   SPTP {A1 7.169, A2 -36.078, A3 70.084, A4 37.543, A5 -95.645, A6 0.000, E1 1384.1, E2 0, E3 0, E4 0, E5 0, E6 0} C_DIS
   SPTP {A1 7.435, A2 -36.403, A3 70.202, A4 38.822, A5 -95.236, A6 0.000, E1 1384.19, E2 0, E3 0, E4 0, E5 0, E6 0} C_DIS
   SPTP {A1 7.436, A2 -36.388, A3 70.184, A4 38.835, A5 -95.248, A6 0.000, E1 1384.17, E2 0, E3 0, E4 0, E5 0, E6 0} C_DIS
   SPTP {A1 7.884, A2 -36.920, A3 70.315, A4 41.034, A5 -94.543, A6 0.000, E1 1384.27, E2 0, E3 0, E4 0, E5 0, E6 0} C_DIS
   SPTP {A1 8.287, A2 -37.697, A3 70.867, A4 43.097, A5 -93.668, A6 0.000, E1 1384.12, E2 0, E3 0, E4 0, E5 0, E6 0} C_DIS
   SPTP {A1 8.650, A2 -38.713, A3 71.817, A4 45.038, A5 -92.609, A6 0.000, E1 1383.69, E2 0, E3 0, E4 0, E5 0, E6 0} C_DIS
   SPTP {A1 9.006, A2 -39.694, A3 72.658, A4 46.997, A5 -91.531, A6 0.000, E1 1383.19, E2 0, E3 0, E4 0, E5 0, E6 0} C_DIS
   SPTP {A1 9.354, A2 -40.644, A3 73.399, A4 48.977, A5 -90.438, A6 0.000, E1 1382.62, E2 0, E3 0, E4 0, E5 0, E6 0} C_DIS
   SPTP {A1 9.691, A2 -41.569, A3 74.056, A4 50.968, A5 -89.331, A6 0.000, E1 1382, E2 0, E3 0, E4 0, E5 0, E6 0} C_DIS
   SPTP {A1 10.017, A2 -42.476, A3 74.643, A4 52.966, A5 -88.208, A6 0.000, E1 1381.33, E2 0, E3 0, E4 0, E5 0, E6 0} C_DIS
   SPTP {A1 10.328, A2 -43.371, A3 75.171, A4 54.967, A5 -87.068, A6 0.000, E1 1380.62, E2 0, E3 0, E4 0, E5 0, E6 0} C_DIS
   SPTP {A1 10.624, A2 -44.257, A3 75.647, A4 56.970, A5 -85.911, A6 0.000, E1 1379.87, E2 0, E3 0, E4 0, E5 0, E6 0} C_DIS
   SPTP {A1 10.880, A2 -45.245, A3 76.287, A4 58.874, A5 -84.671, A6 0.000, E1 1378.9, E2 0, E3 0, E4 0, E5 0, E6 0} C_DIS
   SPTP {A1 11.110, A2 -46.270, A3 76.958, A4 60.747, A5 -83.381, A6 0.000, E1 1377.81, E2 0, E3 0, E4 0, E5 0, E6 0} C_DIS
   SPTP {A1 11.327, A2 -47.266, A3 77.541, A4 62.657, A5 -82.098, A6 0.000, E1 1376.63, E2 0, E3 0, E4 0, E5 0, E6 0} C_DIS
   SPTP {A1 11.525, A2 -48.255, A3 78.076, A4 64.580, A5 -80.798, A6 0.000, E1 1375.41, E2 0, E3 0, E4 0, E5 0, E6 0} C_DIS
   SPTP {A1 11.705, A2 -49.225, A3 78.545, A4 66.533, A5 -79.499, A6 0.000, E1 1374.11, E2 0, E3 0, E4 0, E5 0, E6 0} C_DIS
   SPTP {A1 11.864, A2 -50.188, A3 78.970, A4 68.504, A5 -78.190, A6 0.000, E1 1372.75, E2 0, E3 0, E4 0, E5 0, E6 0} C_DIS
   SPTP {A1 12.001, A2 -51.135, A3 79.340, A4 70.506, A5 -76.884, A6 0.000, E1 1371.32, E2 0, E3 0, E4 0, E5 0, E6 0} C_DIS
   SPTP {A1 12.116, A2 -52.065, A3 79.653, A4 72.544, A5 -75.587, A6 0.000, E1 1369.81, E2 0, E3 0, E4 0, E5 0, E6 0} C_DIS
   SPTP {A1 12.207, A2 -52.982, A3 79.919, A4 74.615, A5 -74.295, A6 0.000, E1 1368.22, E2 0, E3 0, E4 0, E5 0, E6 0} C_DIS
   SPTP {A1 12.274, A2 -53.871, A3 80.119, A4 76.738, A5 -73.033, A6 0.000, E1 1366.55, E2 0, E3 0, E4 0, E5 0, E6 0} C_DIS
   SPTP {A1 12.314, A2 -54.747, A3 80.275, A4 78.900, A5 -71.783, A6 0.000, E1 1364.79, E2 0, E3 0, E4 0, E5 0, E6 0} C_DIS
   SPTP {A1 12.330, A2 -55.585, A3 80.354, A4 81.129, A5 -70.586, A6 0.000, E1 1362.92, E2 0, E3 0, E4 0, E5 0, E6 0} C_DIS
   SPTP {A1 12.318, A2 -56.405, A3 80.388, A4 83.407, A5 -69.414, A6 0.000, E1 1360.97, E2 0, E3 0, E4 0, E5 0, E6 0} C_DIS
   SPTP {A1 12.280, A2 -57.171, A3 80.349, A4 85.710, A5 -68.323, A6 0.000, E1 1358.99, E2 0, E3 0, E4 0, E5 0, E6 0} C_DIS
   SPTP {A1 12.211, A2 -57.855, A3 80.301, A4 87.795, A5 -67.313, A6 0.000, E1 1357.48, E2 0, E3 0, E4 0, E5 0, E6 0} C_DIS
   SPTP {A1 12.118, A2 -58.515, A3 80.224, A4 89.903, A5 -66.338, A6 0.000, E1 1355.95, E2 0, E3 0, E4 0, E5 0, E6 0} C_DIS
   SPTP {A1 12.001, A2 -59.157, A3 80.116, A4 92.058, A5 -65.395, A6 0.000, E1 1354.35, E2 0, E3 0, E4 0, E5 0, E6 0} C_DIS
   SPTP {A1 11.859, A2 -59.776, A3 79.972, A4 94.265, A5 -64.496, A6 0.000, E1 1352.66, E2 0, E3 0, E4 0, E5 0, E6 0} C_DIS
   SPTP {A1 11.695, A2 -60.368, A3 79.786, A4 96.528, A5 -63.651, A6 0.000, E1 1350.9, E2 0, E3 0, E4 0, E5 0, E6 0} C_DIS
   SPTP {A1 11.508, A2 -60.930, A3 79.557, A4 98.848, A5 -62.868, A6 0.000, E1 1349.05, E2 0, E3 0, E4 0, E5 0, E6 0} C_DIS
   SPTP {A1 11.299, A2 -61.454, A3 79.275, A4 101.229, A5 -62.166, A6 0.000, E1 1347.13, E2 0, E3 0, E4 0, E5 0, E6 0} C_DIS
   SPTP {A1 11.071, A2 -61.939, A3 78.958, A4 103.616, A5 -61.537, A6 0.000, E1 1345.24, E2 0, E3 0, E4 0, E5 0, E6 0} C_DIS
   SPTP {A1 10.826, A2 -62.433, A3 78.899, A4 105.464, A5 -60.737, A6 0.000, E1 1344.4, E2 0, E3 0, E4 0, E5 0, E6 0} C_DIS
   SPTP {A1 10.563, A2 -62.914, A3 78.831, A4 107.350, A5 -59.960, A6 0.000, E1 1343.51, E2 0, E3 0, E4 0, E5 0, E6 0} C_DIS
   SPTP {A1 10.285, A2 -63.380, A3 78.749, A4 109.279, A5 -59.216, A6 0.000, E1 1342.58, E2 0, E3 0, E4 0, E5 0, E6 0} C_DIS
   SPTP {A1 9.993, A2 -63.822, A3 78.643, A4 111.251, A5 -58.522, A6 0.000, E1 1341.59, E2 0, E3 0, E4 0, E5 0, E6 0} C_DIS
   SPTP {A1 9.691, A2 -64.237, A3 78.507, A4 113.267, A5 -57.891, A6 0.000, E1 1340.57, E2 0, E3 0, E4 0, E5 0, E6 0} C_DIS
   SPTP {A1 9.380, A2 -64.621, A3 78.337, A4 115.323, A5 -57.335, A6 0.000, E1 1339.52, E2 0, E3 0, E4 0, E5 0, E6 0} C_DIS
   SPTP {A1 9.064, A2 -65.063, A3 78.450, A4 116.938, A5 -56.526, A6 0.000, E1 1339.23, E2 0, E3 0, E4 0, E5 0, E6 0} C_DIS
   SPTP {A1 8.744, A2 -65.577, A3 78.859, A4 118.116, A5 -55.418, A6 0.000, E1 1339.68, E2 0, E3 0, E4 0, E5 0, E6 0} C_DIS
   SPTP {A1 8.422, A2 -66.076, A3 79.265, A4 119.307, A5 -54.327, A6 0.000, E1 1340.12, E2 0, E3 0, E4 0, E5 0, E6 0} C_DIS
   SPTP {A1 8.100, A2 -66.558, A3 79.662, A4 120.507, A5 -53.261, A6 0.000, E1 1340.57, E2 0, E3 0, E4 0, E5 0, E6 0} C_DIS
   SPTP {A1 7.780, A2 -67.022, A3 80.051, A4 121.713, A5 -52.224, A6 0.000, E1 1341.01, E2 0, E3 0, E4 0, E5 0, E6 0} C_DIS
   SPTP {A1 7.467, A2 -67.502, A3 80.560, A4 122.709, A5 -51.073, A6 0.000, E1 1341.77, E2 0, E3 0, E4 0, E5 0, E6 0} C_DIS
   SPTP {A1 7.166, A2 -68.151, A3 81.723, A4 122.565, A5 -49.178, A6 0.000, E1 1344.14, E2 0, E3 0, E4 0, E5 0, E6 0} C_DIS
   SPTP {A1 6.872, A2 -68.768, A3 82.871, A4 122.309, A5 -47.295, A6 0.000, E1 1346.6, E2 0, E3 0, E4 0, E5 0, E6 0} C_DIS
   SPTP {A1 6.589, A2 -69.350, A3 83.999, A4 121.925, A5 -45.437, A6 0.000, E1 1349.17, E2 0, E3 0, E4 0, E5 0, E6 0} C_DIS
   SPTP {A1 6.318, A2 -69.897, A3 85.107, A4 121.400, A5 -43.606, A6 0.000, E1 1351.87, E2 0, E3 0, E4 0, E5 0, E6 0} C_DIS
   SPTP {A1 6.062, A2 -70.438, A3 86.341, A4 120.340, A5 -41.643, A6 0.000, E1 1355.19, E2 0, E3 0, E4 0, E5 0, E6 0} C_DIS
   SPTP {A1 5.824, A2 -71.031, A3 88.135, A4 117.358, A5 -39.081, A6 0.000, E1 1360.71, E2 0, E3 0, E4 0, E5 0, E6 0} C_DIS
   SPTP {A1 5.600, A2 -71.527, A3 89.843, A4 113.809, A5 -36.706, A6 0.000, E1 1366.77, E2 0, E3 0, E4 0, E5 0, E6 0} C_DIS
   SPTP {A1 5.388, A2 -71.926, A3 91.463, A4 109.639, A5 -34.559, A6 0.000, E1 1373.41, E2 0, E3 0, E4 0, E5 0, E6 0} C_DIS
   SPTP {A1 5.188, A2 -72.227, A3 92.993, A4 104.813, A5 -32.690, A6 0.000, E1 1380.66, E2 0, E3 0, E4 0, E5 0, E6 0} C_DIS
   SPTP {A1 5.002, A2 -72.428, A3 94.426, A4 99.341, A5 -31.164, A6 0.000, E1 1388.54, E2 0, E3 0, E4 0, E5 0, E6 0} C_DIS
   SPTP {A1 4.831, A2 -72.507, A3 95.865, A4 92.599, A5 -30.068, A6 0.000, E1 1397.64, E2 0, E3 0, E4 0, E5 0, E6 0} C_DIS
   SPTP {A1 4.667, A2 -72.440, A3 97.273, A4 84.768, A5 -29.571, A6 0.000, E1 1407.76, E2 0, E3 0, E4 0, E5 0, E6 0} C_DIS
   SPTP {A1 4.511, A2 -72.240, A3 98.532, A4 76.835, A5 -29.714, A6 0.000, E1 1417.97, E2 0, E3 0, E4 0, E5 0, E6 0} C_DIS
   SPTP {A1 4.362, A2 -71.911, A3 99.641, A4 69.168, A5 -30.480, A6 0.000, E1 1427.9, E2 0, E3 0, E4 0, E5 0, E6 0} C_DIS
   SPTP {A1 4.222, A2 -71.453, A3 100.593, A4 62.081, A5 -31.820, A6 0.000, E1 1437.23, E2 0, E3 0, E4 0, E5 0, E6 0} C_DIS
   SPTP {A1 4.097, A2 -70.869, A3 101.381, A4 55.785, A5 -33.659, A6 0.000, E1 1445.78, E2 0, E3 0, E4 0, E5 0, E6 0} C_DIS
   SPTP {A1 3.984, A2 -70.165, A3 102.004, A4 50.333, A5 -35.897, A6 0.000, E1 1453.49, E2 0, E3 0, E4 0, E5 0, E6 0} C_DIS
   SPTP {A1 3.885, A2 -69.347, A3 102.462, A4 45.703, A5 -38.442, A6 0.000, E1 1460.39, E2 0, E3 0, E4 0, E5 0, E6 0} C_DIS
   SPTP {A1 3.803, A2 -68.422, A3 102.749, A4 41.834, A5 -41.216, A6 0.000, E1 1466.55, E2 0, E3 0, E4 0, E5 0, E6 0} C_DIS
   SPTP {A1 3.740, A2 -67.451, A3 102.873, A4 38.754, A5 -44.015, A6 0.000, E1 1471.9, E2 0, E3 0, E4 0, E5 0, E6 0} C_DIS
   SPTP {A1 3.689, A2 -66.715, A3 102.919, A4 36.735, A5 -46.135, A6 0.000, E1 1475.93, E2 0, E3 0, E4 0, E5 0, E6 0} C_DIS
   SPTP {A1 3.659, A2 -65.931, A3 102.870, A4 35.037, A5 -48.306, A6 0.000, E1 1479.68, E2 0, E3 0, E4 0, E5 0, E6 0} C_DIS
   SPTP {A1 3.648, A2 -65.104, A3 102.727, A4 33.624, A5 -50.506, A6 0.000, E1 1483.18, E2 0, E3 0, E4 0, E5 0, E6 0} C_DIS
   SPTP {A1 3.657, A2 -64.237, A3 102.492, A4 32.463, A5 -52.721, A6 0.000, E1 1486.45, E2 0, E3 0, E4 0, E5 0, E6 0} C_DIS
   SPTP {A1 3.685, A2 -63.334, A3 102.166, A4 31.531, A5 -54.934, A6 0.000, E1 1489.54, E2 0, E3 0, E4 0, E5 0, E6 0} C_DIS
   SPTP {A1 3.731, A2 -62.398, A3 101.751, A4 30.804, A5 -57.135, A6 0.000, E1 1492.46, E2 0, E3 0, E4 0, E5 0, E6 0} C_DIS
   SPTP {A1 3.826, A2 -61.744, A3 101.405, A4 30.571, A5 -58.666, A6 0.000, E1 1494.88, E2 0, E3 0, E4 0, E5 0, E6 0} C_DIS
   SPTP {A1 3.954, A2 -61.235, A3 101.094, A4 30.616, A5 -59.850, A6 0.000, E1 1497.04, E2 0, E3 0, E4 0, E5 0, E6 0} C_DIS
   SPTP {A1 4.098, A2 -60.718, A3 100.743, A4 30.764, A5 -61.022, A6 0.000, E1 1499.13, E2 0, E3 0, E4 0, E5 0, E6 0} C_DIS
   SPTP {A1 4.257, A2 -60.192, A3 100.353, A4 31.008, A5 -62.179, A6 0.000, E1 1501.14, E2 0, E3 0, E4 0, E5 0, E6 0} C_DIS
   SPTP {A1 4.427, A2 -59.660, A3 99.928, A4 31.331, A5 -63.315, A6 0.000, E1 1503.1, E2 0, E3 0, E4 0, E5 0, E6 0} C_DIS
   SPTP {A1 4.608, A2 -59.122, A3 99.466, A4 31.729, A5 -64.432, A6 0.000, E1 1505.01, E2 0, E3 0, E4 0, E5 0, E6 0} C_DIS
   SPTP {A1 4.798, A2 -58.579, A3 98.969, A4 32.195, A5 -65.525, A6 0.000, E1 1506.87, E2 0, E3 0, E4 0, E5 0, E6 0} C_DIS
   SPTP {A1 4.996, A2 -58.032, A3 98.437, A4 32.722, A5 -66.594, A6 0.000, E1 1508.69, E2 0, E3 0, E4 0, E5 0, E6 0} C_DIS
   SPTP {A1 5.260, A2 -57.817, A3 98.085, A4 33.647, A5 -67.005, A6 0.000, E1 1510.18, E2 0, E3 0, E4 0, E5 0, E6 0} C_DIS
   SPTP {A1 5.539, A2 -57.646, A3 97.738, A4 34.671, A5 -67.316, A6 0.000, E1 1511.58, E2 0, E3 0, E4 0, E5 0, E6 0} C_DIS
   SPTP {A1 5.820, A2 -57.474, A3 97.367, A4 35.734, A5 -67.614, A6 0.000, E1 1512.95, E2 0, E3 0, E4 0, E5 0, E6 0} C_DIS
   SPTP {A1 6.104, A2 -57.298, A3 96.974, A4 36.832, A5 -67.902, A6 0.000, E1 1514.29, E2 0, E3 0, E4 0, E5 0, E6 0} C_DIS
   SPTP {A1 6.390, A2 -57.120, A3 96.557, A4 37.963, A5 -68.180, A6 0.000, E1 1515.59, E2 0, E3 0, E4 0, E5 0, E6 0} C_DIS
   SPTP {A1 6.675, A2 -56.938, A3 96.117, A4 39.121, A5 -68.447, A6 0.000, E1 1516.87, E2 0, E3 0, E4 0, E5 0, E6 0} C_DIS
   SPTP {A1 6.958, A2 -56.755, A3 95.655, A4 40.301, A5 -68.704, A6 0.000, E1 1518.12, E2 0, E3 0, E4 0, E5 0, E6 0} C_DIS
   SPTP {A1 7.239, A2 -56.569, A3 95.173, A4 41.498, A5 -68.950, A6 0.000, E1 1519.36, E2 0, E3 0, E4 0, E5 0, E6 0} C_DIS
   SPTP {A1 7.516, A2 -56.382, A3 94.671, A4 42.710, A5 -69.186, A6 0.000, E1 1520.57, E2 0, E3 0, E4 0, E5 0, E6 0} C_DIS
   SPTP {A1 7.789, A2 -56.194, A3 94.152, A4 43.931, A5 -69.411, A6 0.000, E1 1521.77, E2 0, E3 0, E4 0, E5 0, E6 0} C_DIS
   SPTP {A1 8.056, A2 -56.006, A3 93.616, A4 45.157, A5 -69.624, A6 0.000, E1 1522.95, E2 0, E3 0, E4 0, E5 0, E6 0} C_DIS
   SPTP {A1 8.318, A2 -55.838, A3 93.080, A4 46.408, A5 -69.792, A6 0.000, E1 1524.09, E2 0, E3 0, E4 0, E5 0, E6 0} C_DIS
   SPTP {A1 8.584, A2 -55.773, A3 92.604, A4 47.763, A5 -69.778, A6 0.000, E1 1525.06, E2 0, E3 0, E4 0, E5 0, E6 0} C_DIS
   SPTP {A1 8.843, A2 -55.706, A3 92.111, A4 49.123, A5 -69.759, A6 0.000, E1 1526.02, E2 0, E3 0, E4 0, E5 0, E6 0} C_DIS
   SPTP {A1 9.093, A2 -55.638, A3 91.605, A4 50.483, A5 -69.736, A6 0.000, E1 1526.96, E2 0, E3 0, E4 0, E5 0, E6 0} C_DIS
   SPTP {A1 9.335, A2 -55.569, A3 91.085, A4 51.842, A5 -69.708, A6 0.000, E1 1527.89, E2 0, E3 0, E4 0, E5 0, E6 0} C_DIS
   SPTP {A1 9.568, A2 -55.500, A3 90.556, A4 53.196, A5 -69.675, A6 0.000, E1 1528.82, E2 0, E3 0, E4 0, E5 0, E6 0} C_DIS
   SPTP {A1 9.792, A2 -55.431, A3 90.017, A4 54.545, A5 -69.636, A6 0.000, E1 1529.74, E2 0, E3 0, E4 0, E5 0, E6 0} C_DIS
   SPTP {A1 10.005, A2 -55.365, A3 89.472, A4 55.885, A5 -69.590, A6 0.000, E1 1530.65, E2 0, E3 0, E4 0, E5 0, E6 0} C_DIS
   SPTP {A1 10.208, A2 -55.301, A3 88.922, A4 57.214, A5 -69.538, A6 0.000, E1 1531.57, E2 0, E3 0, E4 0, E5 0, E6 0} C_DIS
   SPTP {A1 10.400, A2 -55.241, A3 88.371, A4 58.530, A5 -69.476, A6 0.000, E1 1532.49, E2 0, E3 0, E4 0, E5 0, E6 0} C_DIS
   SPTP {A1 10.582, A2 -55.186, A3 87.820, A4 59.832, A5 -69.407, A6 0.000, E1 1533.41, E2 0, E3 0, E4 0, E5 0, E6 0} C_DIS
   SPTP {A1 10.740, A2 -55.139, A3 87.304, A4 61.051, A5 -69.348, A6 0.000, E1 1534.31, E2 0, E3 0, E4 0, E5 0, E6 0} C_DIS
   SPTP {A1 10.881, A2 -55.098, A3 86.806, A4 62.225, A5 -69.290, A6 0.000, E1 1535.2, E2 0, E3 0, E4 0, E5 0, E6 0} C_DIS
   SPTP {A1 10.991, A2 -55.067, A3 86.373, A4 63.258, A5 -69.262, A6 0.000, E1 1536.06, E2 0, E3 0, E4 0, E5 0, E6 0} C_DIS
   SPTP {A1 11.093, A2 -55.045, A3 85.951, A4 64.274, A5 -69.222, A6 0.000, E1 1536.93, E2 0, E3 0, E4 0, E5 0, E6 0} C_DIS
   SPTP {A1 11.187, A2 -55.032, A3 85.541, A4 65.272, A5 -69.166, A6 0.000, E1 1537.81, E2 0, E3 0, E4 0, E5 0, E6 0} C_DIS
   SPTP {A1 11.272, A2 -55.031, A3 85.146, A4 66.249, A5 -69.094, A6 0.000, E1 1538.71, E2 0, E3 0, E4 0, E5 0, E6 0} C_DIS
   SPTP {A1 11.348, A2 -55.042, A3 84.767, A4 67.207, A5 -69.004, A6 0.000, E1 1539.62, E2 0, E3 0, E4 0, E5 0, E6 0} C_DIS
   SPTP {A1 11.416, A2 -55.066, A3 84.407, A4 68.144, A5 -68.894, A6 0.000, E1 1540.54, E2 0, E3 0, E4 0, E5 0, E6 0} C_DIS
   SPTP {A1 11.476, A2 -55.104, A3 84.067, A4 69.059, A5 -68.763, A6 0.000, E1 1541.48, E2 0, E3 0, E4 0, E5 0, E6 0} C_DIS
   SPTP {A1 11.528, A2 -55.156, A3 83.748, A4 69.955, A5 -68.611, A6 0.000, E1 1542.44, E2 0, E3 0, E4 0, E5 0, E6 0} C_DIS
   SPTP {A1 11.572, A2 -55.222, A3 83.451, A4 70.830, A5 -68.438, A6 0.000, E1 1543.41, E2 0, E3 0, E4 0, E5 0, E6 0} C_DIS
   SPTP {A1 11.607, A2 -55.304, A3 83.179, A4 71.683, A5 -68.241, A6 0.000, E1 1544.4, E2 0, E3 0, E4 0, E5 0, E6 0} C_DIS
   SPTP {A1 11.635, A2 -55.402, A3 82.932, A4 72.515, A5 -68.020, A6 0.000, E1 1545.4, E2 0, E3 0, E4 0, E5 0, E6 0} C_DIS
   SPTP {A1 11.654, A2 -55.516, A3 82.711, A4 73.326, A5 -67.773, A6 0.000, E1 1546.42, E2 0, E3 0, E4 0, E5 0, E6 0} C_DIS
   SPTP {A1 11.666, A2 -55.648, A3 82.517, A4 74.116, A5 -67.499, A6 0.000, E1 1547.46, E2 0, E3 0, E4 0, E5 0, E6 0} C_DIS
   SPTP {A1 11.669, A2 -55.797, A3 82.353, A4 74.883, A5 -67.197, A6 0.000, E1 1548.51, E2 0, E3 0, E4 0, E5 0, E6 0} C_DIS
   SPTP {A1 11.664, A2 -55.965, A3 82.218, A4 75.628, A5 -66.866, A6 0.000, E1 1549.58, E2 0, E3 0, E4 0, E5 0, E6 0} C_DIS
   SPTP {A1 11.652, A2 -56.149, A3 82.111, A4 76.353, A5 -66.507, A6 0.000, E1 1550.67, E2 0, E3 0, E4 0, E5 0, E6 0} C_DIS
   SPTP {A1 11.630, A2 -56.362, A3 82.047, A4 77.065, A5 -66.113, A6 0.000, E1 1551.69, E2 0, E3 0, E4 0, E5 0, E6 0} C_DIS
   SPTP {A1 11.594, A2 -56.634, A3 82.059, A4 77.786, A5 -65.663, A6 0.000, E1 1552.49, E2 0, E3 0, E4 0, E5 0, E6 0} C_DIS
   SPTP {A1 11.550, A2 -56.917, A3 82.090, A4 78.495, A5 -65.192, A6 0.000, E1 1553.28, E2 0, E3 0, E4 0, E5 0, E6 0} C_DIS
   SPTP {A1 11.500, A2 -57.212, A3 82.142, A4 79.190, A5 -64.698, A6 0.000, E1 1554.09, E2 0, E3 0, E4 0, E5 0, E6 0} C_DIS
   SPTP {A1 11.441, A2 -57.521, A3 82.216, A4 79.870, A5 -64.178, A6 0.000, E1 1554.9, E2 0, E3 0, E4 0, E5 0, E6 0} C_DIS
   SPTP {A1 11.376, A2 -57.842, A3 82.311, A4 80.536, A5 -63.633, A6 0.000, E1 1555.72, E2 0, E3 0, E4 0, E5 0, E6 0} C_DIS
   SPTP {A1 11.303, A2 -58.175, A3 82.427, A4 81.187, A5 -63.061, A6 0.000, E1 1556.54, E2 0, E3 0, E4 0, E5 0, E6 0} C_DIS
   SPTP {A1 11.221, A2 -58.523, A3 82.567, A4 81.823, A5 -62.460, A6 0.000, E1 1557.37, E2 0, E3 0, E4 0, E5 0, E6 0} C_DIS
   SPTP {A1 11.132, A2 -58.883, A3 82.729, A4 82.445, A5 -61.830, A6 0.000, E1 1558.21, E2 0, E3 0, E4 0, E5 0, E6 0} C_DIS
   SPTP {A1 11.034, A2 -59.254, A3 82.911, A4 83.052, A5 -61.173, A6 0.000, E1 1559.05, E2 0, E3 0, E4 0, E5 0, E6 0} C_DIS
   SPTP {A1 10.928, A2 -59.638, A3 83.113, A4 83.646, A5 -60.488, A6 0.000, E1 1559.89, E2 0, E3 0, E4 0, E5 0, E6 0} C_DIS
   SPTP {A1 10.814, A2 -60.032, A3 83.335, A4 84.226, A5 -59.773, A6 0.000, E1 1560.74, E2 0, E3 0, E4 0, E5 0, E6 0} C_DIS
   SPTP {A1 10.694, A2 -60.461, A3 83.535, A4 84.991, A5 -58.980, A6 0.000, E1 1561.36, E2 0, E3 0, E4 0, E5 0, E6 0} C_DIS
   SPTP {A1 10.569, A2 -60.935, A3 83.675, A4 86.092, A5 -58.086, A6 0.000, E1 1561.6, E2 0, E3 0, E4 0, E5 0, E6 0} C_DIS
   SPTP {A1 10.434, A2 -61.410, A3 83.815, A4 87.208, A5 -57.183, A6 0.000, E1 1561.81, E2 0, E3 0, E4 0, E5 0, E6 0} C_DIS
   SPTP {A1 10.286, A2 -61.889, A3 83.966, A4 88.333, A5 -56.260, A6 0.000, E1 1561.99, E2 0, E3 0, E4 0, E5 0, E6 0} C_DIS
   SPTP {A1 10.126, A2 -62.369, A3 84.121, A4 89.474, A5 -55.324, A6 0.000, E1 1562.14, E2 0, E3 0, E4 0, E5 0, E6 0} C_DIS
   SPTP {A1 9.955, A2 -62.849, A3 84.279, A4 90.632, A5 -54.376, A6 0.000, E1 1562.27, E2 0, E3 0, E4 0, E5 0, E6 0} C_DIS
   SPTP {A1 9.772, A2 -63.328, A3 84.441, A4 91.811, A5 -53.418, A6 0.000, E1 1562.36, E2 0, E3 0, E4 0, E5 0, E6 0} C_DIS
   SPTP {A1 9.577, A2 -63.807, A3 84.606, A4 93.011, A5 -52.448, A6 0.000, E1 1562.42, E2 0, E3 0, E4 0, E5 0, E6 0} C_DIS
   SPTP {A1 9.369, A2 -64.286, A3 84.774, A4 94.235, A5 -51.467, A6 0.000, E1 1562.44, E2 0, E3 0, E4 0, E5 0, E6 0} C_DIS
   SPTP {A1 9.150, A2 -64.762, A3 84.944, A4 95.486, A5 -50.477, A6 0.000, E1 1562.42, E2 0, E3 0, E4 0, E5 0, E6 0} C_DIS
   SPTP {A1 8.919, A2 -65.236, A3 85.116, A4 96.767, A5 -49.479, A6 0.000, E1 1562.37, E2 0, E3 0, E4 0, E5 0, E6 0} C_DIS
   SPTP {A1 8.675, A2 -65.707, A3 85.289, A4 98.082, A5 -48.474, A6 0.000, E1 1562.26, E2 0, E3 0, E4 0, E5 0, E6 0} C_DIS
   SPTP {A1 8.419, A2 -66.174, A3 85.463, A4 99.433, A5 -47.462, A6 0.000, E1 1562.11, E2 0, E3 0, E4 0, E5 0, E6 0} C_DIS
   SPTP {A1 8.152, A2 -66.637, A3 85.636, A4 100.824, A5 -46.448, A6 0.000, E1 1561.9, E2 0, E3 0, E4 0, E5 0, E6 0} C_DIS
   SPTP {A1 7.872, A2 -67.094, A3 85.809, A4 102.261, A5 -45.431, A6 0.000, E1 1561.65, E2 0, E3 0, E4 0, E5 0, E6 0} C_DIS
   SPTP {A1 7.572, A2 -67.552, A3 85.912, A4 104.037, A5 -44.369, A6 0.000, E1 1561.18, E2 0, E3 0, E4 0, E5 0, E6 0} C_DIS
   SPTP {A1 7.252, A2 -68.004, A3 85.969, A4 106.070, A5 -43.290, A6 0.000, E1 1560.53, E2 0, E3 0, E4 0, E5 0, E6 0} C_DIS
   SPTP {A1 6.917, A2 -68.445, A3 86.023, A4 108.181, A5 -42.230, A6 0.000, E1 1559.8, E2 0, E3 0, E4 0, E5 0, E6 0} C_DIS
   SPTP {A1 6.567, A2 -68.876, A3 86.074, A4 110.377, A5 -41.192, A6 0.000, E1 1558.98, E2 0, E3 0, E4 0, E5 0, E6 0} C_DIS
   SPTP {A1 6.203, A2 -69.294, A3 86.121, A4 112.662, A5 -40.181, A6 0.000, E1 1558.06, E2 0, E3 0, E4 0, E5 0, E6 0} C_DIS
   SPTP {A1 5.826, A2 -69.699, A3 86.164, A4 115.041, A5 -39.202, A6 0.000, E1 1557.04, E2 0, E3 0, E4 0, E5 0, E6 0} C_DIS
   SPTP {A1 5.437, A2 -70.089, A3 86.201, A4 117.516, A5 -38.264, A6 0.000, E1 1555.92, E2 0, E3 0, E4 0, E5 0, E6 0} C_DIS
   SPTP {A1 5.038, A2 -70.464, A3 86.231, A4 120.087, A5 -37.373, A6 0.000, E1 1554.7, E2 0, E3 0, E4 0, E5 0, E6 0} C_DIS
   SPTP {A1 4.629, A2 -70.822, A3 86.254, A4 122.755, A5 -36.536, A6 0.000, E1 1553.39, E2 0, E3 0, E4 0, E5 0, E6 0} C_DIS
   SPTP {A1 4.213, A2 -71.164, A3 86.270, A4 125.515, A5 -35.759, A6 0.000, E1 1551.99, E2 0, E3 0, E4 0, E5 0, E6 0} C_DIS
   SPTP {A1 3.791, A2 -71.489, A3 86.280, A4 128.361, A5 -35.048, A6 0.000, E1 1550.51, E2 0, E3 0, E4 0, E5 0, E6 0} C_DIS
   SPTP {A1 3.362, A2 -71.797, A3 86.284, A4 131.289, A5 -34.401, A6 0.000, E1 1548.95, E2 0, E3 0, E4 0, E5 0, E6 0} C_DIS
   SPTP {A1 2.929, A2 -72.089, A3 86.283, A4 134.283, A5 -33.830, A6 0.000, E1 1547.34, E2 0, E3 0, E4 0, E5 0, E6 0} C_DIS
   SPTP {A1 2.497, A2 -72.363, A3 86.275, A4 137.326, A5 -33.340, A6 0.000, E1 1545.69, E2 0, E3 0, E4 0, E5 0, E6 0} C_DIS
   SPTP {A1 2.061, A2 -72.738, A3 86.699, A4 139.518, A5 -32.220, A6 0.000, E1 1545.11, E2 0, E3 0, E4 0, E5 0, E6 0} C_DIS
   SPTP {A1 1.627, A2 -73.105, A3 87.145, A4 141.756, A5 -31.099, A6 0.000, E1 1544.5, E2 0, E3 0, E4 0, E5 0, E6 0} C_DIS
   SPTP {A1 1.197, A2 -73.461, A3 87.598, A4 144.072, A5 -30.003, A6 0.000, E1 1543.81, E2 0, E3 0, E4 0, E5 0, E6 0} C_DIS
   SPTP {A1 0.774, A2 -73.805, A3 88.058, A4 146.455, A5 -28.939, A6 0.000, E1 1543.06, E2 0, E3 0, E4 0, E5 0, E6 0} C_DIS
   SPTP {A1 0.364, A2 -74.137, A3 88.523, A4 148.889, A5 -27.913, A6 0.000, E1 1542.28, E2 0, E3 0, E4 0, E5 0, E6 0} C_DIS
   SPTP {A1 -0.030, A2 -74.457, A3 88.993, A4 151.354, A5 -26.928, A6 0.000, E1 1541.49, E2 0, E3 0, E4 0, E5 0, E6 0} C_DIS
   SPTP {A1 -0.405, A2 -74.766, A3 89.471, A4 153.826, A5 -25.983, A6 0.000, E1 1540.72, E2 0, E3 0, E4 0, E5 0, E6 0} C_DIS
   SPTP {A1 -0.746, A2 -75.184, A3 90.489, A4 155.098, A5 -24.066, A6 0.000, E1 1541.17, E2 0, E3 0, E4 0, E5 0, E6 0} C_DIS
   SPTP {A1 -1.054, A2 -75.610, A3 91.676, A4 155.848, A5 -21.809, A6 0.000, E1 1542.15, E2 0, E3 0, E4 0, E5 0, E6 0} C_DIS
   SPTP {A1 -1.331, A2 -76.002, A3 92.847, A4 156.441, A5 -19.554, A6 0.000, E1 1543.3, E2 0, E3 0, E4 0, E5 0, E6 0} C_DIS
   SPTP {A1 -1.568, A2 -76.358, A3 93.998, A4 156.735, A5 -17.311, A6 0.000, E1 1544.77, E2 0, E3 0, E4 0, E5 0, E6 0} C_DIS
   SPTP {A1 -1.756, A2 -76.678, A3 95.128, A4 156.518, A5 -15.091, A6 0.000, E1 1546.78, E2 0, E3 0, E4 0, E5 0, E6 0} C_DIS
   SPTP {A1 -1.896, A2 -76.995, A3 96.809, A4 152.367, A5 -11.592, A6 0.000, E1 1552.7, E2 0, E3 0, E4 0, E5 0, E6 0} C_DIS
   SPTP {A1 -1.981, A2 -77.209, A3 98.592, A4 141.183, A5 -7.873, A6 0.000, E1 1565.64, E2 0, E3 0, E4 0, E5 0, E6 0} C_DIS
   SPTP {A1 -2.021, A2 -77.294, A3 100.256, A4 112.941, A5 -5.050, A6 0.000, E1 1595.64, E2 0, E3 0, E4 0, E5 0, E6 0} C_DIS
   SPTP {A1 -2.002, A2 -77.248, A3 101.792, A4 64.079, A5 -5.073, A6 0.000, E1 1646.28, E2 0, E3 0, E4 0, E5 0, E6 0} C_DIS
   SPTP {A1 -1.933, A2 -77.002, A3 103.360, A4 33.430, A5 -8.458, A6 0.000, E1 1678.73, E2 0, E3 0, E4 0, E5 0, E6 0} C_DIS
   SPTP {A1 -1.835, A2 -76.340, A3 105.094, A4 19.922, A5 -14.412, A6 0.000, E1 1694.04, E2 0, E3 0, E4 0, E5 0, E6 0} C_DIS
   SPTP {A1 -1.691, A2 -75.378, A3 106.478, A4 15.024, A5 -20.704, A6 0.000, E1 1700.74, E2 0, E3 0, E4 0, E5 0, E6 0} C_DIS
   SPTP {A1 -1.523, A2 -74.130, A3 107.499, A4 12.755, A5 -27.040, A6 0.000, E1 1704.8, E2 0, E3 0, E4 0, E5 0, E6 0} C_DIS
   SPTP {A1 -1.336, A2 -72.048, A3 108.206, A4 10.956, A5 -35.192, A6 0.000, E1 1708.67, E2 0, E3 0, E4 0, E5 0, E6 0} C_DIS
   SPTP {A1 -1.139, A2 -69.470, A3 108.247, A4 10.032, A5 -43.410, A6 0.000, E1 1711.71, E2 0, E3 0, E4 0, E5 0, E6 0} C_DIS
   SPTP {A1 -0.943, A2 -66.541, A3 107.588, A4 9.626, A5 -51.310, A6 0.000, E1 1714.26, E2 0, E3 0, E4 0, E5 0, E6 0} C_DIS
   SPTP {A1 -0.760, A2 -63.337, A3 106.239, A4 9.484, A5 -58.805, A6 0.000, E1 1716.57, E2 0, E3 0, E4 0, E5 0, E6 0} C_DIS
   SPTP {A1 -0.402, A2 -60.558, A3 104.609, A4 10.067, A5 -64.621, A6 0.000, E1 1718.92, E2 0, E3 0, E4 0, E5 0, E6 0} C_DIS
   SPTP {A1 0.021, A2 -57.871, A3 102.654, A4 10.957, A5 -69.737, A6 0.000, E1 1721.27, E2 0, E3 0, E4 0, E5 0, E6 0} C_DIS
   SPTP {A1 0.459, A2 -55.144, A3 100.310, A4 11.991, A5 -74.482, A6 0.000, E1 1723.57, E2 0, E3 0, E4 0, E5 0, E6 0} C_DIS
   SPTP {A1 0.910, A2 -52.403, A3 97.596, A4 13.172, A5 -78.847, A6 0.000, E1 1725.84, E2 0, E3 0, E4 0, E5 0, E6 0} C_DIS
   SPTP {A1 1.366, A2 -49.664, A3 94.532, A4 14.469, A5 -82.826, A6 0.000, E1 1728.09, E2 0, E3 0, E4 0, E5 0, E6 0} C_DIS
   SPTP {A1 1.826, A2 -46.935, A3 91.129, A4 15.883, A5 -86.424, A6 0.000, E1 1730.31, E2 0, E3 0, E4 0, E5 0, E6 0} C_DIS
   SPTP {A1 2.292, A2 -44.215, A3 87.387, A4 17.435, A5 -89.652, A6 0.000, E1 1732.48, E2 0, E3 0, E4 0, E5 0, E6 0} C_DIS
   SPTP {A1 2.759, A2 -41.494, A3 83.304, A4 19.102, A5 -92.517, A6 0.000, E1 1734.6, E2 0, E3 0, E4 0, E5 0, E6 0} C_DIS
   SPTP {A1 3.224, A2 -38.757, A3 78.863, A4 20.878, A5 -95.028, A6 0.000, E1 1736.63, E2 0, E3 0, E4 0, E5 0, E6 0} C_DIS
   SPTP {A1 3.682, A2 -35.973, A3 74.027, A4 22.751, A5 -97.192, A6 0.000, E1 1738.54, E2 0, E3 0, E4 0, E5 0, E6 0} C_DIS
   SPTP {A1 4.205, A2 -34.811, A3 71.616, A4 24.821, A5 -97.894, A6 0.000, E1 1740.06, E2 0, E3 0, E4 0, E5 0, E6 0} C_DIS
   SPTP {A1 4.770, A2 -34.693, A3 70.859, A4 27.041, A5 -97.795, A6 0.000, E1 1741.24, E2 0, E3 0, E4 0, E5 0, E6 0} C_DIS
   SPTP {A1 5.325, A2 -34.554, A3 70.010, A4 29.319, A5 -97.666, A6 0.000, E1 1742.28, E2 0, E3 0, E4 0, E5 0, E6 0} C_DIS
   SPTP {A1 5.867, A2 -34.386, A3 69.065, A4 31.639, A5 -97.513, A6 0.000, E1 1743.18, E2 0, E3 0, E4 0, E5 0, E6 0} C_DIS
   SPTP {A1 6.350, A2 -35.016, A3 69.499, A4 33.767, A5 -96.859, A6 0.000, E1 1743.63, E2 0, E3 0, E4 0, E5 0, E6 0} C_DIS
   SPTP {A1 6.822, A2 -35.633, A3 69.868, A4 35.924, A5 -96.173, A6 0.000, E1 1743.93, E2 0, E3 0, E4 0, E5 0, E6 0} C_DIS
   SPTP {A1 7.132, A2 -36.019, A3 70.050, A4 37.375, A5 -95.712, A6 0.000, E1 1744.07, E2 0, E3 0, E4 0, E5 0, E6 0} C_DIS
   SPTP {A1 7.436, A2 -36.388, A3 70.184, A4 38.835, A5 -95.248, A6 0.000, E1 1744.17, E2 0, E3 0, E4 0, E5 0, E6 0} C_DIS
   SPTP {A1 7.437, A2 -36.374, A3 70.166, A4 38.848, A5 -95.259, A6 0.000, E1 1744.15, E2 0, E3 0, E4 0, E5 0, E6 0} C_DIS
   SPTP {A1 7.885, A2 -36.902, A3 70.292, A4 41.049, A5 -94.557, A6 0.000, E1 1744.24, E2 0, E3 0, E4 0, E5 0, E6 0} C_DIS
   SPTP {A1 8.288, A2 -37.675, A3 70.838, A4 43.114, A5 -93.685, A6 0.000, E1 1744.09, E2 0, E3 0, E4 0, E5 0, E6 0} C_DIS
   SPTP {A1 8.652, A2 -38.689, A3 71.784, A4 45.058, A5 -92.630, A6 0.000, E1 1743.66, E2 0, E3 0, E4 0, E5 0, E6 0} C_DIS
   SPTP {A1 9.007, A2 -39.668, A3 72.623, A4 47.017, A5 -91.554, A6 0.000, E1 1743.16, E2 0, E3 0, E4 0, E5 0, E6 0} C_DIS
   SPTP {A1 9.356, A2 -40.617, A3 73.362, A4 48.999, A5 -90.462, A6 0.000, E1 1742.59, E2 0, E3 0, E4 0, E5 0, E6 0} C_DIS
   SPTP {A1 9.693, A2 -41.541, A3 74.018, A4 50.990, A5 -89.358, A6 0.000, E1 1741.97, E2 0, E3 0, E4 0, E5 0, E6 0} C_DIS
   SPTP {A1 10.018, A2 -42.447, A3 74.603, A4 52.989, A5 -88.237, A6 0.000, E1 1741.3, E2 0, E3 0, E4 0, E5 0, E6 0} C_DIS
   SPTP {A1 10.330, A2 -43.341, A3 75.130, A4 54.990, A5 -87.099, A6 0.000, E1 1740.59, E2 0, E3 0, E4 0, E5 0, E6 0} C_DIS
   SPTP {A1 10.626, A2 -44.225, A3 75.605, A4 56.993, A5 -85.944, A6 0.000, E1 1739.84, E2 0, E3 0, E4 0, E5 0, E6 0} C_DIS
   SPTP {A1 10.882, A2 -45.212, A3 76.244, A4 58.898, A5 -84.707, A6 0.000, E1 1738.87, E2 0, E3 0, E4 0, E5 0, E6 0} C_DIS
   SPTP {A1 11.113, A2 -46.237, A3 76.915, A4 60.772, A5 -83.419, A6 0.000, E1 1737.78, E2 0, E3 0, E4 0, E5 0, E6 0} C_DIS
   SPTP {A1 11.330, A2 -47.232, A3 77.497, A4 62.683, A5 -82.138, A6 0.000, E1 1736.61, E2 0, E3 0, E4 0, E5 0, E6 0} C_DIS
   SPTP {A1 11.529, A2 -48.221, A3 78.032, A4 64.605, A5 -80.840, A6 0.000, E1 1735.38, E2 0, E3 0, E4 0, E5 0, E6 0} C_DIS
   SPTP {A1 11.709, A2 -49.191, A3 78.502, A4 66.558, A5 -79.543, A6 0.000, E1 1734.08, E2 0, E3 0, E4 0, E5 0, E6 0} C_DIS
   SPTP {A1 11.868, A2 -50.153, A3 78.927, A4 68.529, A5 -78.235, A6 0.000, E1 1732.73, E2 0, E3 0, E4 0, E5 0, E6 0} C_DIS
   SPTP {A1 12.006, A2 -51.101, A3 79.297, A4 70.530, A5 -76.930, A6 0.000, E1 1731.3, E2 0, E3 0, E4 0, E5 0, E6 0} C_DIS
   SPTP {A1 12.121, A2 -52.031, A3 79.611, A4 72.567, A5 -75.635, A6 0.000, E1 1729.79, E2 0, E3 0, E4 0, E5 0, E6 0} C_DIS
   SPTP {A1 12.212, A2 -52.947, A3 79.878, A4 74.637, A5 -74.344, A6 0.000, E1 1728.21, E2 0, E3 0, E4 0, E5 0, E6 0} C_DIS
   SPTP {A1 12.279, A2 -53.837, A3 80.079, A4 76.759, A5 -73.083, A6 0.000, E1 1726.53, E2 0, E3 0, E4 0, E5 0, E6 0} C_DIS
   SPTP {A1 12.319, A2 -54.713, A3 80.236, A4 78.920, A5 -71.834, A6 0.000, E1 1724.78, E2 0, E3 0, E4 0, E5 0, E6 0} C_DIS
   SPTP {A1 12.336, A2 -55.551, A3 80.316, A4 81.147, A5 -70.637, A6 0.000, E1 1722.91, E2 0, E3 0, E4 0, E5 0, E6 0} C_DIS
   SPTP {A1 12.324, A2 -56.372, A3 80.352, A4 83.422, A5 -69.466, A6 0.000, E1 1720.96, E2 0, E3 0, E4 0, E5 0, E6 0} C_DIS
   SPTP {A1 12.286, A2 -57.139, A3 80.314, A4 85.723, A5 -68.374, A6 0.000, E1 1718.99, E2 0, E3 0, E4 0, E5 0, E6 0} C_DIS
   SPTP {A1 12.217, A2 -57.824, A3 80.268, A4 87.807, A5 -67.364, A6 0.000, E1 1717.48, E2 0, E3 0, E4 0, E5 0, E6 0} C_DIS
   SPTP {A1 12.125, A2 -58.485, A3 80.192, A4 89.913, A5 -66.389, A6 0.000, E1 1715.95, E2 0, E3 0, E4 0, E5 0, E6 0} C_DIS
   SPTP {A1 12.008, A2 -59.127, A3 80.086, A4 92.065, A5 -65.446, A6 0.000, E1 1714.35, E2 0, E3 0, E4 0, E5 0, E6 0} C_DIS
   SPTP {A1 11.867, A2 -59.748, A3 79.944, A4 94.269, A5 -64.546, A6 0.000, E1 1712.67, E2 0, E3 0, E4 0, E5 0, E6 0} C_DIS
   SPTP {A1 11.703, A2 -60.340, A3 79.760, A4 96.529, A5 -63.700, A6 0.000, E1 1710.91, E2 0, E3 0, E4 0, E5 0, E6 0} C_DIS
   SPTP {A1 11.515, A2 -60.904, A3 79.534, A4 98.846, A5 -62.915, A6 0.000, E1 1709.07, E2 0, E3 0, E4 0, E5 0, E6 0} C_DIS
   SPTP {A1 11.307, A2 -61.430, A3 79.254, A4 101.223, A5 -62.210, A6 0.000, E1 1707.15, E2 0, E3 0, E4 0, E5 0, E6 0} C_DIS
   SPTP {A1 11.079, A2 -61.916, A3 78.938, A4 103.611, A5 -61.581, A6 0.000, E1 1705.25, E2 0, E3 0, E4 0, E5 0, E6 0} C_DIS
   SPTP {A1 10.833, A2 -62.411, A3 78.881, A4 105.456, A5 -60.778, A6 0.000, E1 1704.42, E2 0, E3 0, E4 0, E5 0, E6 0} C_DIS
   SPTP {A1 10.571, A2 -62.894, A3 78.816, A4 107.339, A5 -59.998, A6 0.000, E1 1703.53, E2 0, E3 0, E4 0, E5 0, E6 0} C_DIS
   SPTP {A1 10.292, A2 -63.361, A3 78.736, A4 109.265, A5 -59.251, A6 0.000, E1 1702.6, E2 0, E3 0, E4 0, E5 0, E6 0} C_DIS
   SPTP {A1 10.001, A2 -63.805, A3 78.633, A4 111.234, A5 -58.554, A6 0.000, E1 1701.62, E2 0, E3 0, E4 0, E5 0, E6 0} C_DIS
   SPTP {A1 9.698, A2 -64.222, A3 78.500, A4 113.247, A5 -57.920, A6 0.000, E1 1700.6, E2 0, E3 0, E4 0, E5 0, E6 0} C_DIS
   SPTP {A1 9.387, A2 -64.607, A3 78.333, A4 115.301, A5 -57.360, A6 0.000, E1 1699.54, E2 0, E3 0, E4 0, E5 0, E6 0} C_DIS
   SPTP {A1 9.071, A2 -65.049, A3 78.442, A4 116.922, A5 -56.553, A6 0.000, E1 1699.24, E2 0, E3 0, E4 0, E5 0, E6 0} C_DIS
   SPTP {A1 8.750, A2 -65.565, A3 78.854, A4 118.099, A5 -55.441, A6 0.000, E1 1699.69, E2 0, E3 0, E4 0, E5 0, E6 0} C_DIS
   SPTP {A1 8.428, A2 -66.066, A3 79.262, A4 119.287, A5 -54.346, A6 0.000, E1 1700.13, E2 0, E3 0, E4 0, E5 0, E6 0} C_DIS
   SPTP {A1 8.105, A2 -66.550, A3 79.662, A4 120.486, A5 -53.276, A6 0.000, E1 1700.57, E2 0, E3 0, E4 0, E5 0, E6 0} C_DIS
   SPTP {A1 7.785, A2 -67.015, A3 80.053, A4 121.692, A5 -52.235, A6 0.000, E1 1701.01, E2 0, E3 0, E4 0, E5 0, E6 0} C_DIS
   SPTP {A1 7.471, A2 -67.494, A3 80.553, A4 122.705, A5 -51.094, A6 0.000, E1 1701.75, E2 0, E3 0, E4 0, E5 0, E6 0} C_DIS
   SPTP {A1 7.169, A2 -68.144, A3 81.716, A4 122.563, A5 -49.196, A6 0.000, E1 1704.11, E2 0, E3 0, E4 0, E5 0, E6 0} C_DIS
   SPTP {A1 6.875, A2 -68.761, A3 82.865, A4 122.310, A5 -47.311, A6 0.000, E1 1706.56, E2 0, E3 0, E4 0, E5 0, E6 0} C_DIS
   SPTP {A1 6.590, A2 -69.345, A3 83.994, A4 121.929, A5 -45.450, A6 0.000, E1 1709.12, E2 0, E3 0, E4 0, E5 0, E6 0} C_DIS
   SPTP {A1 6.317, A2 -69.893, A3 85.102, A4 121.408, A5 -43.616, A6 0.000, E1 1711.82, E2 0, E3 0, E4 0, E5 0, E6 0} C_DIS
   SPTP {A1 6.060, A2 -70.432, A3 86.322, A4 120.389, A5 -41.667, A6 0.000, E1 1715.08, E2 0, E3 0, E4 0, E5 0, E6 0} C_DIS
   SPTP {A1 5.822, A2 -71.027, A3 88.116, A4 117.421, A5 -39.101, A6 0.000, E1 1720.59, E2 0, E3 0, E4 0, E5 0, E6 0} C_DIS
   SPTP {A1 5.596, A2 -71.525, A3 89.824, A4 113.887, A5 -36.721, A6 0.000, E1 1726.62, E2 0, E3 0, E4 0, E5 0, E6 0} C_DIS
   SPTP {A1 5.383, A2 -71.926, A3 91.445, A4 109.733, A5 -34.567, A6 0.000, E1 1733.24, E2 0, E3 0, E4 0, E5 0, E6 0} C_DIS
   SPTP {A1 5.182, A2 -72.229, A3 92.976, A4 104.924, A5 -32.689, A6 0.000, E1 1740.48, E2 0, E3 0, E4 0, E5 0, E6 0} C_DIS
   SPTP {A1 4.995, A2 -72.433, A3 94.410, A4 99.467, A5 -31.154, A6 0.000, E1 1748.34, E2 0, E3 0, E4 0, E5 0, E6 0} C_DIS
   SPTP {A1 4.823, A2 -72.515, A3 95.844, A4 92.773, A5 -30.046, A6 0.000, E1 1757.38, E2 0, E3 0, E4 0, E5 0, E6 0} C_DIS
   SPTP {A1 4.659, A2 -72.452, A3 97.254, A4 84.948, A5 -29.532, A6 0.000, E1 1767.5, E2 0, E3 0, E4 0, E5 0, E6 0} C_DIS
   SPTP {A1 4.502, A2 -72.257, A3 98.516, A4 77.011, A5 -29.658, A6 0.000, E1 1777.71, E2 0, E3 0, E4 0, E5 0, E6 0} C_DIS
   SPTP {A1 4.352, A2 -71.931, A3 99.627, A4 69.330, A5 -30.407, A6 0.000, E1 1787.65, E2 0, E3 0, E4 0, E5 0, E6 0} C_DIS
   SPTP {A1 4.213, A2 -71.478, A3 100.583, A4 62.225, A5 -31.732, A6 0.000, E1 1797, E2 0, E3 0, E4 0, E5 0, E6 0} C_DIS
   SPTP {A1 4.087, A2 -70.898, A3 101.374, A4 55.905, A5 -33.558, A6 0.000, E1 1805.57, E2 0, E3 0, E4 0, E5 0, E6 0} C_DIS
   SPTP {A1 3.974, A2 -70.198, A3 102.002, A4 50.435, A5 -35.786, A6 0.000, E1 1813.29, E2 0, E3 0, E4 0, E5 0, E6 0} C_DIS
   SPTP {A1 3.875, A2 -69.385, A3 102.464, A4 45.785, A5 -38.321, A6 0.000, E1 1820.21, E2 0, E3 0, E4 0, E5 0, E6 0} C_DIS
   SPTP {A1 3.794, A2 -68.465, A3 102.757, A4 41.899, A5 -41.088, A6 0.000, E1 1826.38, E2 0, E3 0, E4 0, E5 0, E6 0} C_DIS
   SPTP {A1 3.731, A2 -67.484, A3 102.884, A4 38.776, A5 -43.917, A6 0.000, E1 1831.78, E2 0, E3 0, E4 0, E5 0, E6 0} C_DIS
   SPTP {A1 3.680, A2 -66.750, A3 102.933, A4 36.753, A5 -46.035, A6 0.000, E1 1835.82, E2 0, E3 0, E4 0, E5 0, E6 0} C_DIS
   SPTP {A1 3.650, A2 -65.968, A3 102.887, A4 35.051, A5 -48.204, A6 0.000, E1 1839.57, E2 0, E3 0, E4 0, E5 0, E6 0} C_DIS
   SPTP {A1 3.640, A2 -65.143, A3 102.747, A4 33.632, A5 -50.404, A6 0.000, E1 1843.07, E2 0, E3 0, E4 0, E5 0, E6 0} C_DIS
   SPTP {A1 3.648, A2 -64.278, A3 102.516, A4 32.466, A5 -52.617, A6 0.000, E1 1846.35, E2 0, E3 0, E4 0, E5 0, E6 0} C_DIS
   SPTP {A1 3.676, A2 -63.377, A3 102.194, A4 31.531, A5 -54.830, A6 0.000, E1 1849.43, E2 0, E3 0, E4 0, E5 0, E6 0} C_DIS
   SPTP {A1 3.723, A2 -62.443, A3 101.782, A4 30.803, A5 -57.031, A6 0.000, E1 1852.35, E2 0, E3 0, E4 0, E5 0, E6 0} C_DIS
   SPTP {A1 3.816, A2 -61.768, A3 101.427, A4 30.546, A5 -58.609, A6 0.000, E1 1854.8, E2 0, E3 0, E4 0, E5 0, E6 0} C_DIS
   SPTP {A1 3.943, A2 -61.260, A3 101.118, A4 30.589, A5 -59.793, A6 0.000, E1 1856.96, E2 0, E3 0, E4 0, E5 0, E6 0} C_DIS
   SPTP {A1 4.087, A2 -60.742, A3 100.769, A4 30.736, A5 -60.966, A6 0.000, E1 1859.04, E2 0, E3 0, E4 0, E5 0, E6 0} C_DIS
   SPTP {A1 4.246, A2 -60.217, A3 100.380, A4 30.980, A5 -62.123, A6 0.000, E1 1861.06, E2 0, E3 0, E4 0, E5 0, E6 0} C_DIS
   SPTP {A1 4.416, A2 -59.685, A3 99.956, A4 31.301, A5 -63.260, A6 0.000, E1 1863.02, E2 0, E3 0, E4 0, E5 0, E6 0} C_DIS
   SPTP {A1 4.597, A2 -59.148, A3 99.496, A4 31.697, A5 -64.377, A6 0.000, E1 1864.92, E2 0, E3 0, E4 0, E5 0, E6 0} C_DIS
   SPTP {A1 4.787, A2 -58.605, A3 99.000, A4 32.163, A5 -65.472, A6 0.000, E1 1866.78, E2 0, E3 0, E4 0, E5 0, E6 0} C_DIS
   SPTP {A1 4.985, A2 -58.058, A3 98.470, A4 32.689, A5 -66.542, A6 0.000, E1 1868.6, E2 0, E3 0, E4 0, E5 0, E6 0} C_DIS
   SPTP {A1 5.245, A2 -57.822, A3 98.107, A4 33.590, A5 -66.993, A6 0.000, E1 1870.1, E2 0, E3 0, E4 0, E5 0, E6 0} C_DIS
   SPTP {A1 5.523, A2 -57.652, A3 97.760, A4 34.613, A5 -67.305, A6 0.000, E1 1871.51, E2 0, E3 0, E4 0, E5 0, E6 0} C_DIS
   SPTP {A1 5.805, A2 -57.479, A3 97.391, A4 35.675, A5 -67.605, A6 0.000, E1 1872.88, E2 0, E3 0, E4 0, E5 0, E6 0} C_DIS
   SPTP {A1 6.089, A2 -57.303, A3 96.998, A4 36.771, A5 -67.893, A6 0.000, E1 1874.21, E2 0, E3 0, E4 0, E5 0, E6 0} C_DIS
   SPTP {A1 6.374, A2 -57.125, A3 96.582, A4 37.901, A5 -68.171, A6 0.000, E1 1875.52, E2 0, E3 0, E4 0, E5 0, E6 0} C_DIS
   SPTP {A1 6.659, A2 -56.944, A3 96.143, A4 39.057, A5 -68.440, A6 0.000, E1 1876.8, E2 0, E3 0, E4 0, E5 0, E6 0} C_DIS
   SPTP {A1 6.943, A2 -56.760, A3 95.683, A4 40.236, A5 -68.697, A6 0.000, E1 1878.05, E2 0, E3 0, E4 0, E5 0, E6 0} C_DIS
   SPTP {A1 7.224, A2 -56.574, A3 95.202, A4 41.432, A5 -68.945, A6 0.000, E1 1879.28, E2 0, E3 0, E4 0, E5 0, E6 0} C_DIS
   SPTP {A1 7.501, A2 -56.387, A3 94.701, A4 42.642, A5 -69.181, A6 0.000, E1 1880.49, E2 0, E3 0, E4 0, E5 0, E6 0} C_DIS
   SPTP {A1 7.774, A2 -56.198, A3 94.182, A4 43.863, A5 -69.407, A6 0.000, E1 1881.69, E2 0, E3 0, E4 0, E5 0, E6 0} C_DIS
   SPTP {A1 8.041, A2 -56.010, A3 93.648, A4 45.088, A5 -69.621, A6 0.000, E1 1882.87, E2 0, E3 0, E4 0, E5 0, E6 0} C_DIS
   SPTP {A1 8.302, A2 -55.835, A3 93.107, A4 46.329, A5 -69.803, A6 0.000, E1 1884.03, E2 0, E3 0, E4 0, E5 0, E6 0} C_DIS
   SPTP {A1 8.569, A2 -55.770, A3 92.632, A4 47.683, A5 -69.789, A6 0.000, E1 1884.99, E2 0, E3 0, E4 0, E5 0, E6 0} C_DIS
   SPTP {A1 8.828, A2 -55.703, A3 92.141, A4 49.041, A5 -69.771, A6 0.000, E1 1885.95, E2 0, E3 0, E4 0, E5 0, E6 0} C_DIS
   SPTP {A1 9.079, A2 -55.635, A3 91.636, A4 50.400, A5 -69.748, A6 0.000, E1 1886.89, E2 0, E3 0, E4 0, E5 0, E6 0} C_DIS
   SPTP {A1 9.321, A2 -55.566, A3 91.117, A4 51.758, A5 -69.720, A6 0.000, E1 1887.82, E2 0, E3 0, E4 0, E5 0, E6 0} C_DIS
   SPTP {A1 9.554, A2 -55.497, A3 90.589, A4 53.111, A5 -69.687, A6 0.000, E1 1888.75, E2 0, E3 0, E4 0, E5 0, E6 0} C_DIS
   SPTP {A1 9.778, A2 -55.428, A3 90.051, A4 54.459, A5 -69.649, A6 0.000, E1 1889.67, E2 0, E3 0, E4 0, E5 0, E6 0} C_DIS
   SPTP {A1 9.992, A2 -55.362, A3 89.507, A4 55.798, A5 -69.604, A6 0.000, E1 1890.59, E2 0, E3 0, E4 0, E5 0, E6 0} C_DIS
   SPTP {A1 10.196, A2 -55.298, A3 88.958, A4 57.127, A5 -69.552, A6 0.000, E1 1891.5, E2 0, E3 0, E4 0, E5 0, E6 0} C_DIS
   SPTP {A1 10.388, A2 -55.238, A3 88.407, A4 58.442, A5 -69.491, A6 0.000, E1 1892.42, E2 0, E3 0, E4 0, E5 0, E6 0} C_DIS
   SPTP {A1 10.571, A2 -55.182, A3 87.856, A4 59.745, A5 -69.422, A6 0.000, E1 1893.34, E2 0, E3 0, E4 0, E5 0, E6 0} C_DIS
   SPTP {A1 10.730, A2 -55.135, A3 87.338, A4 60.968, A5 -69.363, A6 0.000, E1 1894.24, E2 0, E3 0, E4 0, E5 0, E6 0} C_DIS
   SPTP {A1 10.874, A2 -55.094, A3 86.836, A4 62.154, A5 -69.302, A6 0.000, E1 1895.14, E2 0, E3 0, E4 0, E5 0, E6 0} C_DIS
   SPTP {A1 10.985, A2 -55.062, A3 86.403, A4 63.187, A5 -69.275, A6 0.000, E1 1895.99, E2 0, E3 0, E4 0, E5 0, E6 0} C_DIS
   SPTP {A1 11.087, A2 -55.040, A3 85.980, A4 64.202, A5 -69.235, A6 0.000, E1 1896.86, E2 0, E3 0, E4 0, E5 0, E6 0} C_DIS
   SPTP {A1 11.181, A2 -55.026, A3 85.569, A4 65.200, A5 -69.180, A6 0.000, E1 1897.74, E2 0, E3 0, E4 0, E5 0, E6 0} C_DIS
   SPTP {A1 11.266, A2 -55.024, A3 85.174, A4 66.178, A5 -69.109, A6 0.000, E1 1898.64, E2 0, E3 0, E4 0, E5 0, E6 0} C_DIS
   SPTP {A1 11.344, A2 -55.034, A3 84.794, A4 67.136, A5 -69.020, A6 0.000, E1 1899.55, E2 0, E3 0, E4 0, E5 0, E6 0} C_DIS
   SPTP {A1 11.412, A2 -55.057, A3 84.432, A4 68.075, A5 -68.912, A6 0.000, E1 1900.47, E2 0, E3 0, E4 0, E5 0, E6 0} C_DIS
   SPTP {A1 11.473, A2 -55.094, A3 84.092, A4 68.991, A5 -68.782, A6 0.000, E1 1901.41, E2 0, E3 0, E4 0, E5 0, E6 0} C_DIS
   SPTP {A1 11.525, A2 -55.145, A3 83.772, A4 69.887, A5 -68.632, A6 0.000, E1 1902.36, E2 0, E3 0, E4 0, E5 0, E6 0} C_DIS
   SPTP {A1 11.569, A2 -55.210, A3 83.473, A4 70.762, A5 -68.461, A6 0.000, E1 1903.33, E2 0, E3 0, E4 0, E5 0, E6 0} C_DIS
   SPTP {A1 11.605, A2 -55.291, A3 83.199, A4 71.617, A5 -68.266, A6 0.000, E1 1904.32, E2 0, E3 0, E4 0, E5 0, E6 0} C_DIS
   SPTP {A1 11.634, A2 -55.387, A3 82.950, A4 72.450, A5 -68.046, A6 0.000, E1 1905.32, E2 0, E3 0, E4 0, E5 0, E6 0} C_DIS
   SPTP {A1 11.654, A2 -55.500, A3 82.727, A4 73.262, A5 -67.802, A6 0.000, E1 1906.34, E2 0, E3 0, E4 0, E5 0, E6 0} C_DIS
   SPTP {A1 11.666, A2 -55.630, A3 82.531, A4 74.053, A5 -67.531, A6 0.000, E1 1907.37, E2 0, E3 0, E4 0, E5 0, E6 0} C_DIS
   SPTP {A1 11.670, A2 -55.777, A3 82.364, A4 74.821, A5 -67.233, A6 0.000, E1 1908.42, E2 0, E3 0, E4 0, E5 0, E6 0} C_DIS
   SPTP {A1 11.666, A2 -55.943, A3 82.226, A4 75.568, A5 -66.905, A6 0.000, E1 1909.49, E2 0, E3 0, E4 0, E5 0, E6 0} C_DIS
   SPTP {A1 11.654, A2 -56.126, A3 82.118, A4 76.294, A5 -66.548, A6 0.000, E1 1910.57, E2 0, E3 0, E4 0, E5 0, E6 0} C_DIS
   SPTP {A1 11.634, A2 -56.333, A3 82.045, A4 77.005, A5 -66.159, A6 0.000, E1 1911.63, E2 0, E3 0, E4 0, E5 0, E6 0} C_DIS
   SPTP {A1 11.598, A2 -56.604, A3 82.056, A4 77.726, A5 -65.712, A6 0.000, E1 1912.42, E2 0, E3 0, E4 0, E5 0, E6 0} C_DIS
   SPTP {A1 11.555, A2 -56.885, A3 82.085, A4 78.436, A5 -65.244, A6 0.000, E1 1913.22, E2 0, E3 0, E4 0, E5 0, E6 0} C_DIS
   SPTP {A1 11.505, A2 -57.179, A3 82.134, A4 79.132, A5 -64.752, A6 0.000, E1 1914.02, E2 0, E3 0, E4 0, E5 0, E6 0} C_DIS
   SPTP {A1 11.448, A2 -57.486, A3 82.206, A4 79.813, A5 -64.235, A6 0.000, E1 1914.83, E2 0, E3 0, E4 0, E5 0, E6 0} C_DIS
   SPTP {A1 11.383, A2 -57.806, A3 82.299, A4 80.480, A5 -63.693, A6 0.000, E1 1915.65, E2 0, E3 0, E4 0, E5 0, E6 0} C_DIS
   SPTP {A1 11.311, A2 -58.138, A3 82.413, A4 81.133, A5 -63.125, A6 0.000, E1 1916.47, E2 0, E3 0, E4 0, E5 0, E6 0} C_DIS
   SPTP {A1 11.231, A2 -58.483, A3 82.550, A4 81.770, A5 -62.528, A6 0.000, E1 1917.3, E2 0, E3 0, E4 0, E5 0, E6 0} C_DIS
   SPTP {A1 11.142, A2 -58.840, A3 82.708, A4 82.393, A5 -61.903, A6 0.000, E1 1918.13, E2 0, E3 0, E4 0, E5 0, E6 0} C_DIS
   SPTP {A1 11.046, A2 -59.211, A3 82.888, A4 83.002, A5 -61.250, A6 0.000, E1 1918.97, E2 0, E3 0, E4 0, E5 0, E6 0} C_DIS
   SPTP {A1 10.941, A2 -59.592, A3 83.088, A4 83.597, A5 -60.568, A6 0.000, E1 1919.82, E2 0, E3 0, E4 0, E5 0, E6 0} C_DIS
   SPTP {A1 10.827, A2 -59.985, A3 83.308, A4 84.178, A5 -59.857, A6 0.000, E1 1920.66, E2 0, E3 0, E4 0, E5 0, E6 0} C_DIS
   SPTP {A1 10.708, A2 -60.407, A3 83.516, A4 84.894, A5 -59.080, A6 0.000, E1 1921.34, E2 0, E3 0, E4 0, E5 0, E6 0} C_DIS
   SPTP {A1 10.584, A2 -60.881, A3 83.655, A4 85.993, A5 -58.188, A6 0.000, E1 1921.58, E2 0, E3 0, E4 0, E5 0, E6 0} C_DIS
   SPTP {A1 10.450, A2 -61.355, A3 83.796, A4 87.106, A5 -57.286, A6 0.000, E1 1921.79, E2 0, E3 0, E4 0, E5 0, E6 0} C_DIS
   SPTP {A1 10.303, A2 -61.834, A3 83.945, A4 88.230, A5 -56.366, A6 0.000, E1 1921.98, E2 0, E3 0, E4 0, E5 0, E6 0} C_DIS
   SPTP {A1 10.145, A2 -62.313, A3 84.100, A4 89.368, A5 -55.432, A6 0.000, E1 1922.14, E2 0, E3 0, E4 0, E5 0, E6 0} C_DIS
   SPTP {A1 9.975, A2 -62.793, A3 84.257, A4 90.524, A5 -54.488, A6 0.000, E1 1922.26, E2 0, E3 0, E4 0, E5 0, E6 0} C_DIS
   SPTP {A1 9.794, A2 -63.272, A3 84.418, A4 91.700, A5 -53.532, A6 0.000, E1 1922.36, E2 0, E3 0, E4 0, E5 0, E6 0} C_DIS
   SPTP {A1 9.600, A2 -63.750, A3 84.582, A4 92.897, A5 -52.565, A6 0.000, E1 1922.42, E2 0, E3 0, E4 0, E5 0, E6 0} C_DIS
   SPTP {A1 9.395, A2 -64.228, A3 84.750, A4 94.118, A5 -51.587, A6 0.000, E1 1922.45, E2 0, E3 0, E4 0, E5 0, E6 0} C_DIS
   SPTP {A1 9.177, A2 -64.704, A3 84.920, A4 95.365, A5 -50.599, A6 0.000, E1 1922.44, E2 0, E3 0, E4 0, E5 0, E6 0} C_DIS
   SPTP {A1 8.947, A2 -65.178, A3 85.091, A4 96.642, A5 -49.603, A6 0.000, E1 1922.38, E2 0, E3 0, E4 0, E5 0, E6 0} C_DIS
   SPTP {A1 8.705, A2 -65.649, A3 85.264, A4 97.952, A5 -48.599, A6 0.000, E1 1922.28, E2 0, E3 0, E4 0, E5 0, E6 0} C_DIS
   SPTP {A1 8.451, A2 -66.117, A3 85.438, A4 99.297, A5 -47.589, A6 0.000, E1 1922.14, E2 0, E3 0, E4 0, E5 0, E6 0} C_DIS
   SPTP {A1 8.185, A2 -66.579, A3 85.612, A4 100.683, A5 -46.576, A6 0.000, E1 1921.94, E2 0, E3 0, E4 0, E5 0, E6 0} C_DIS
   SPTP {A1 7.907, A2 -67.037, A3 85.785, A4 102.113, A5 -45.561, A6 0.000, E1 1921.69, E2 0, E3 0, E4 0, E5 0, E6 0} C_DIS
   SPTP {A1 7.610, A2 -67.494, A3 85.899, A4 103.833, A5 -44.508, A6 0.000, E1 1921.25, E2 0, E3 0, E4 0, E5 0, E6 0} C_DIS
   SPTP {A1 7.292, A2 -67.947, A3 85.957, A4 105.854, A5 -43.429, A6 0.000, E1 1920.62, E2 0, E3 0, E4 0, E5 0, E6 0} C_DIS
   SPTP {A1 6.959, A2 -68.389, A3 86.011, A4 107.954, A5 -42.369, A6 0.000, E1 1919.9, E2 0, E3 0, E4 0, E5 0, E6 0} C_DIS
   SPTP {A1 6.611, A2 -68.821, A3 86.063, A4 110.137, A5 -41.328, A6 0.000, E1 1919.09, E2 0, E3 0, E4 0, E5 0, E6 0} C_DIS
   SPTP {A1 6.249, A2 -69.240, A3 86.111, A4 112.409, A5 -40.315, A6 0.000, E1 1918.18, E2 0, E3 0, E4 0, E5 0, E6 0} C_DIS
   SPTP {A1 5.874, A2 -69.647, A3 86.155, A4 114.773, A5 -39.331, A6 0.000, E1 1917.18, E2 0, E3 0, E4 0, E5 0, E6 0} C_DIS
   SPTP {A1 5.487, A2 -70.040, A3 86.193, A4 117.234, A5 -38.388, A6 0.000, E1 1916.07, E2 0, E3 0, E4 0, E5 0, E6 0} C_DIS
   SPTP {A1 5.089, A2 -70.416, A3 86.225, A4 119.791, A5 -37.491, A6 0.000, E1 1914.87, E2 0, E3 0, E4 0, E5 0, E6 0} C_DIS
   SPTP {A1 4.682, A2 -70.777, A3 86.249, A4 122.444, A5 -36.648, A6 0.000, E1 1913.57, E2 0, E3 0, E4 0, E5 0, E6 0} C_DIS
   SPTP {A1 4.266, A2 -71.121, A3 86.267, A4 125.191, A5 -35.863, A6 0.000, E1 1912.18, E2 0, E3 0, E4 0, E5 0, E6 0} C_DIS
   SPTP {A1 3.845, A2 -71.447, A3 86.278, A4 128.023, A5 -35.143, A6 0.000, E1 1910.71, E2 0, E3 0, E4 0, E5 0, E6 0} C_DIS
   SPTP {A1 3.416, A2 -71.758, A3 86.284, A4 130.939, A5 -34.488, A6 0.000, E1 1909.17, E2 0, E3 0, E4 0, E5 0, E6 0} C_DIS
   SPTP {A1 2.984, A2 -72.052, A3 86.284, A4 133.924, A5 -33.905, A6 0.000, E1 1907.56, E2 0, E3 0, E4 0, E5 0, E6 0} C_DIS
   SPTP {A1 2.551, A2 -72.329, A3 86.277, A4 136.960, A5 -33.404, A6 0.000, E1 1905.92, E2 0, E3 0, E4 0, E5 0, E6 0} C_DIS
   SPTP {A1 2.116, A2 -72.692, A3 86.653, A4 139.244, A5 -32.357, A6 0.000, E1 1905.22, E2 0, E3 0, E4 0, E5 0, E6 0} C_DIS
   SPTP {A1 1.681, A2 -73.061, A3 87.099, A4 141.471, A5 -31.232, A6 0.000, E1 1904.61, E2 0, E3 0, E4 0, E5 0, E6 0} C_DIS
   SPTP {A1 1.250, A2 -73.419, A3 87.551, A4 143.777, A5 -30.132, A6 0.000, E1 1903.93, E2 0, E3 0, E4 0, E5 0, E6 0} C_DIS
   SPTP {A1 0.826, A2 -73.765, A3 88.011, A4 146.155, A5 -29.061, A6 0.000, E1 1903.18, E2 0, E3 0, E4 0, E5 0, E6 0} C_DIS
   SPTP {A1 0.413, A2 -74.098, A3 88.476, A4 148.587, A5 -28.028, A6 0.000, E1 1902.4, E2 0, E3 0, E4 0, E5 0, E6 0} C_DIS
   SPTP {A1 0.016, A2 -74.420, A3 88.946, A4 151.052, A5 -27.036, A6 0.000, E1 1901.6, E2 0, E3 0, E4 0, E5 0, E6 0} C_DIS
   SPTP {A1 -0.361, A2 -74.730, A3 89.422, A4 153.528, A5 -26.085, A6 0.000, E1 1900.82, E2 0, E3 0, E4 0, E5 0, E6 0} C_DIS
   SPTP {A1 -0.709, A2 -75.132, A3 90.357, A4 154.998, A5 -24.321, A6 0.000, E1 1901.07, E2 0, E3 0, E4 0, E5 0, E6 0} C_DIS
   SPTP {A1 -1.022, A2 -75.562, A3 91.546, A4 155.778, A5 -22.062, A6 0.000, E1 1902.01, E2 0, E3 0, E4 0, E5 0, E6 0} C_DIS
   SPTP {A1 -1.305, A2 -75.958, A3 92.717, A4 156.407, A5 -19.807, A6 0.000, E1 1903.12, E2 0, E3 0, E4 0, E5 0, E6 0} C_DIS
   SPTP {A1 -1.550, A2 -76.318, A3 93.871, A4 156.780, A5 -17.559, A6 0.000, E1 1904.5, E2 0, E3 0, E4 0, E5 0, E6 0} C_DIS
   SPTP {A1 -1.745, A2 -76.642, A3 95.002, A4 156.660, A5 -15.337, A6 0.000, E1 1906.41, E2 0, E3 0, E4 0, E5 0, E6 0} C_DIS
   SPTP {A1 -1.894, A2 -76.961, A3 96.593, A4 153.316, A5 -12.042, A6 0.000, E1 1911.52, E2 0, E3 0, E4 0, E5 0, E6 0} C_DIS
   SPTP {A1 -1.989, A2 -77.190, A3 98.388, A4 143.349, A5 -8.267, A6 0.000, E1 1923.24, E2 0, E3 0, E4 0, E5 0, E6 0} C_DIS
   SPTP {A1 -2.037, A2 -77.291, A3 100.065, A4 118.164, A5 -5.242, A6 0.000, E1 1950.18, E2 0, E3 0, E4 0, E5 0, E6 0} C_DIS
   SPTP {A1 -2.027, A2 -77.261, A3 101.615, A4 69.275, A5 -4.816, A6 0.000, E1 2000.84, E2 0, E3 0, E4 0, E5 0, E6 0} C_DIS
   SPTP {A1 -1.966, A2 -77.064, A3 103.126, A4 36.174, A5 -7.742, A6 0.000, E1 2035.73, E2 0, E3 0, E4 0, E5 0, E6 0} C_DIS
   SPTP {A1 -1.874, A2 -76.442, A3 104.900, A4 20.629, A5 -13.606, A6 0.000, E1 2053.07, E2 0, E3 0, E4 0, E5 0, E6 0} C_DIS
   SPTP {A1 -1.736, A2 -75.519, A3 106.327, A4 15.217, A5 -19.875, A6 0.000, E1 2060.28, E2 0, E3 0, E4 0, E5 0, E6 0} C_DIS
   SPTP {A1 -1.573, A2 -74.309, A3 107.395, A4 12.766, A5 -26.205, A6 0.000, E1 2064.52, E2 0, E3 0, E4 0, E5 0, E6 0} C_DIS
   SPTP {A1 -1.391, A2 -72.359, A3 108.158, A4 10.960, A5 -34.078, A6 0.000, E1 2068.35, E2 0, E3 0, E4 0, E5 0, E6 0} C_DIS
   SPTP {A1 -1.193, A2 -69.840, A3 108.291, A4 9.977, A5 -42.316, A6 0.000, E1 2071.45, E2 0, E3 0, E4 0, E5 0, E6 0} C_DIS
   SPTP {A1 -0.996, A2 -66.960, A3 107.729, A4 9.533, A5 -50.250, A6 0.000, E1 2074.03, E2 0, E3 0, E4 0, E5 0, E6 0} C_DIS
   SPTP {A1 -0.809, A2 -63.795, A3 106.477, A4 9.379, A5 -57.791, A6 0.000, E1 2076.34, E2 0, E3 0, E4 0, E5 0, E6 0} C_DIS
   SPTP {A1 -0.483, A2 -60.933, A3 104.863, A4 9.857, A5 -63.870, A6 0.000, E1 2078.66, E2 0, E3 0, E4 0, E5 0, E6 0} C_DIS
   SPTP {A1 -0.060, A2 -58.259, A3 102.968, A4 10.735, A5 -69.028, A6 0.000, E1 2081, E2 0, E3 0, E4 0, E5 0, E6 0} C_DIS
   SPTP {A1 0.377, A2 -55.542, A3 100.685, A4 11.754, A5 -73.819, A6 0.000, E1 2083.31, E2 0, E3 0, E4 0, E5 0, E6 0} C_DIS
   SPTP {A1 0.829, A2 -52.807, A3 98.030, A4 12.924, A5 -78.231, A6 0.000, E1 2085.56, E2 0, E3 0, E4 0, E5 0, E6 0} C_DIS
   SPTP {A1 1.287, A2 -50.072, A3 95.022, A4 14.215, A5 -82.259, A6 0.000, E1 2087.8, E2 0, E3 0, E4 0, E5 0, E6 0} C_DIS
   SPTP {A1 1.748, A2 -47.348, A3 91.676, A4 15.619, A5 -85.907, A6 0.000, E1 2090.02, E2 0, E3 0, E4 0, E5 0, E6 0} C_DIS
   SPTP {A1 2.215, A2 -44.632, A3 87.993, A4 17.156, A5 -89.184, A6 0.000, E1 2092.19, E2 0, E3 0, E4 0, E5 0, E6 0} C_DIS
   SPTP {A1 2.683, A2 -41.916, A3 83.969, A4 18.813, A5 -92.099, A6 0.000, E1 2094.31, E2 0, E3 0, E4 0, E5 0, E6 0} C_DIS
   SPTP {A1 3.149, A2 -39.189, A3 79.594, A4 20.575, A5 -94.660, A6 0.000, E1 2096.35, E2 0, E3 0, E4 0, E5 0, E6 0} C_DIS
   SPTP {A1 3.609, A2 -36.418, A3 74.829, A4 22.439, A5 -96.875, A6 0.000, E1 2098.27, E2 0, E3 0, E4 0, E5 0, E6 0} C_DIS
   SPTP {A1 4.114, A2 -34.828, A3 71.737, A4 24.466, A5 -97.910, A6 0.000, E1 2099.87, E2 0, E3 0, E4 0, E5 0, E6 0} C_DIS
   SPTP {A1 4.679, A2 -34.712, A3 70.992, A4 26.677, A5 -97.817, A6 0.000, E1 2101.07, E2 0, E3 0, E4 0, E5 0, E6 0} C_DIS
   SPTP {A1 5.236, A2 -34.574, A3 70.155, A4 28.949, A5 -97.693, A6 0.000, E1 2102.12, E2 0, E3 0, E4 0, E5 0, E6 0} C_DIS
   SPTP {A1 5.780, A2 -34.409, A3 69.222, A4 31.264, A5 -97.545, A6 0.000, E1 2103.04, E2 0, E3 0, E4 0, E5 0, E6 0} C_DIS
   SPTP {A1 6.272, A2 -34.903, A3 69.421, A4 33.425, A5 -96.977, A6 0.000, E1 2103.56, E2 0, E3 0, E4 0, E5 0, E6 0} C_DIS
   SPTP {A1 6.746, A2 -35.524, A3 69.805, A4 35.577, A5 -96.295, A6 0.000, E1 2103.88, E2 0, E3 0, E4 0, E5 0, E6 0} C_DIS
   SPTP {A1 7.095, A2 -35.960, A3 70.016, A4 37.207, A5 -95.779, A6 0.000, E1 2104.04, E2 0, E3 0, E4 0, E5 0, E6 0} C_DIS
   SPTP {A1 7.437, A2 -36.374, A3 70.166, A4 38.848, A5 -95.259, A6 0.000, E1 2104.15, E2 0, E3 0, E4 0, E5 0, E6 0} C_DIS
   SPTP {A1 7.438, A2 -36.359, A3 70.148, A4 38.862, A5 -95.271, A6 0.000, E1 2104.13, E2 0, E3 0, E4 0, E5 0, E6 0} C_DIS
   SPTP {A1 7.885, A2 -36.884, A3 70.269, A4 41.063, A5 -94.571, A6 0.000, E1 2104.22, E2 0, E3 0, E4 0, E5 0, E6 0} C_DIS
   SPTP {A1 8.289, A2 -37.654, A3 70.810, A4 43.131, A5 -93.702, A6 0.000, E1 2104.06, E2 0, E3 0, E4 0, E5 0, E6 0} C_DIS
   SPTP {A1 8.653, A2 -38.665, A3 71.751, A4 45.077, A5 -92.650, A6 0.000, E1 2103.63, E2 0, E3 0, E4 0, E5 0, E6 0} C_DIS
   SPTP {A1 9.009, A2 -39.643, A3 72.588, A4 47.038, A5 -91.576, A6 0.000, E1 2103.12, E2 0, E3 0, E4 0, E5 0, E6 0} C_DIS
   SPTP {A1 9.357, A2 -40.590, A3 73.326, A4 49.020, A5 -90.487, A6 0.000, E1 2102.56, E2 0, E3 0, E4 0, E5 0, E6 0} C_DIS
   SPTP {A1 9.695, A2 -41.513, A3 73.979, A4 51.012, A5 -89.385, A6 0.000, E1 2101.93, E2 0, E3 0, E4 0, E5 0, E6 0} C_DIS
   SPTP {A1 10.020, A2 -42.418, A3 74.563, A4 53.011, A5 -88.267, A6 0.000, E1 2101.26, E2 0, E3 0, E4 0, E5 0, E6 0} C_DIS
   SPTP {A1 10.332, A2 -43.311, A3 75.090, A4 55.013, A5 -87.131, A6 0.000, E1 2100.55, E2 0, E3 0, E4 0, E5 0, E6 0} C_DIS
   SPTP {A1 10.628, A2 -44.194, A3 75.564, A4 57.016, A5 -85.978, A6 0.000, E1 2099.81, E2 0, E3 0, E4 0, E5 0, E6 0} C_DIS
   SPTP {A1 10.885, A2 -45.180, A3 76.200, A4 58.922, A5 -84.743, A6 0.000, E1 2098.84, E2 0, E3 0, E4 0, E5 0, E6 0} C_DIS
   SPTP {A1 11.116, A2 -46.204, A3 76.871, A4 60.796, A5 -83.457, A6 0.000, E1 2097.75, E2 0, E3 0, E4 0, E5 0, E6 0} C_DIS
   SPTP {A1 11.333, A2 -47.198, A3 77.453, A4 62.708, A5 -82.179, A6 0.000, E1 2096.58, E2 0, E3 0, E4 0, E5 0, E6 0} C_DIS
   SPTP {A1 11.532, A2 -48.187, A3 77.988, A4 64.630, A5 -80.881, A6 0.000, E1 2095.35, E2 0, E3 0, E4 0, E5 0, E6 0} C_DIS
   SPTP {A1 11.713, A2 -49.157, A3 78.458, A4 66.582, A5 -79.586, A6 0.000, E1 2094.06, E2 0, E3 0, E4 0, E5 0, E6 0} C_DIS
   SPTP {A1 11.872, A2 -50.119, A3 78.884, A4 68.553, A5 -78.280, A6 0.000, E1 2092.7, E2 0, E3 0, E4 0, E5 0, E6 0} C_DIS
   SPTP {A1 12.010, A2 -51.067, A3 79.255, A4 70.553, A5 -76.976, A6 0.000, E1 2091.28, E2 0, E3 0, E4 0, E5 0, E6 0} C_DIS
   SPTP {A1 12.125, A2 -51.996, A3 79.569, A4 72.590, A5 -75.682, A6 0.000, E1 2089.77, E2 0, E3 0, E4 0, E5 0, E6 0} C_DIS
   SPTP {A1 12.216, A2 -52.913, A3 79.837, A4 74.659, A5 -74.393, A6 0.000, E1 2088.19, E2 0, E3 0, E4 0, E5 0, E6 0} C_DIS
   SPTP {A1 12.284, A2 -53.803, A3 80.038, A4 76.779, A5 -73.133, A6 0.000, E1 2086.52, E2 0, E3 0, E4 0, E5 0, E6 0} C_DIS
   SPTP {A1 12.325, A2 -54.679, A3 80.196, A4 78.939, A5 -71.885, A6 0.000, E1 2084.76, E2 0, E3 0, E4 0, E5 0, E6 0} C_DIS
   SPTP {A1 12.342, A2 -55.518, A3 80.278, A4 81.165, A5 -70.689, A6 0.000, E1 2082.91, E2 0, E3 0, E4 0, E5 0, E6 0} C_DIS
   SPTP {A1 12.330, A2 -56.339, A3 80.315, A4 83.438, A5 -69.518, A6 0.000, E1 2080.96, E2 0, E3 0, E4 0, E5 0, E6 0} C_DIS
   SPTP {A1 12.292, A2 -57.107, A3 80.279, A4 85.737, A5 -68.426, A6 0.000, E1 2078.98, E2 0, E3 0, E4 0, E5 0, E6 0} C_DIS
   SPTP {A1 12.224, A2 -57.793, A3 80.235, A4 87.819, A5 -67.415, A6 0.000, E1 2077.48, E2 0, E3 0, E4 0, E5 0, E6 0} C_DIS
   SPTP {A1 12.131, A2 -58.454, A3 80.160, A4 89.922, A5 -66.440, A6 0.000, E1 2075.96, E2 0, E3 0, E4 0, E5 0, E6 0} C_DIS
   SPTP {A1 12.015, A2 -59.098, A3 80.056, A4 92.072, A5 -65.496, A6 0.000, E1 2074.36, E2 0, E3 0, E4 0, E5 0, E6 0} C_DIS
   SPTP {A1 11.874, A2 -59.719, A3 79.915, A4 94.273, A5 -64.596, A6 0.000, E1 2072.68, E2 0, E3 0, E4 0, E5 0, E6 0} C_DIS
   SPTP {A1 11.710, A2 -60.313, A3 79.734, A4 96.530, A5 -63.749, A6 0.000, E1 2070.92, E2 0, E3 0, E4 0, E5 0, E6 0} C_DIS
   SPTP {A1 11.523, A2 -60.878, A3 79.510, A4 98.843, A5 -62.961, A6 0.000, E1 2069.09, E2 0, E3 0, E4 0, E5 0, E6 0} C_DIS
   SPTP {A1 11.315, A2 -61.405, A3 79.233, A4 101.217, A5 -62.254, A6 0.000, E1 2067.17, E2 0, E3 0, E4 0, E5 0, E6 0} C_DIS
   SPTP {A1 11.087, A2 -61.893, A3 78.918, A4 103.606, A5 -61.624, A6 0.000, E1 2065.27, E2 0, E3 0, E4 0, E5 0, E6 0} C_DIS
   SPTP {A1 10.841, A2 -62.389, A3 78.863, A4 105.448, A5 -60.819, A6 0.000, E1 2064.43, E2 0, E3 0, E4 0, E5 0, E6 0} C_DIS
   SPTP {A1 10.579, A2 -62.873, A3 78.800, A4 107.328, A5 -60.037, A6 0.000, E1 2063.55, E2 0, E3 0, E4 0, E5 0, E6 0} C_DIS
   SPTP {A1 10.300, A2 -63.342, A3 78.723, A4 109.251, A5 -59.287, A6 0.000, E1 2062.62, E2 0, E3 0, E4 0, E5 0, E6 0} C_DIS
   SPTP {A1 10.008, A2 -63.788, A3 78.623, A4 111.217, A5 -58.586, A6 0.000, E1 2061.64, E2 0, E3 0, E4 0, E5 0, E6 0} C_DIS
   SPTP {A1 9.705, A2 -64.207, A3 78.493, A4 113.227, A5 -57.948, A6 0.000, E1 2060.62, E2 0, E3 0, E4 0, E5 0, E6 0} C_DIS
   SPTP {A1 9.394, A2 -64.594, A3 78.329, A4 115.278, A5 -57.384, A6 0.000, E1 2059.57, E2 0, E3 0, E4 0, E5 0, E6 0} C_DIS
   SPTP {A1 9.078, A2 -65.036, A3 78.434, A4 116.907, A5 -56.580, A6 0.000, E1 2059.25, E2 0, E3 0, E4 0, E5 0, E6 0} C_DIS
   SPTP {A1 8.757, A2 -65.554, A3 78.849, A4 118.081, A5 -55.464, A6 0.000, E1 2059.7, E2 0, E3 0, E4 0, E5 0, E6 0} C_DIS
   SPTP {A1 8.434, A2 -66.057, A3 79.259, A4 119.268, A5 -54.365, A6 0.000, E1 2060.14, E2 0, E3 0, E4 0, E5 0, E6 0} C_DIS
   SPTP {A1 8.111, A2 -66.542, A3 79.662, A4 120.466, A5 -53.291, A6 0.000, E1 2060.58, E2 0, E3 0, E4 0, E5 0, E6 0} C_DIS
   SPTP {A1 7.790, A2 -67.008, A3 80.055, A4 121.671, A5 -52.247, A6 0.000, E1 2061.02, E2 0, E3 0, E4 0, E5 0, E6 0} C_DIS
   SPTP {A1 7.475, A2 -67.485, A3 80.545, A4 122.701, A5 -51.114, A6 0.000, E1 2061.72, E2 0, E3 0, E4 0, E5 0, E6 0} C_DIS
   SPTP {A1 7.172, A2 -68.136, A3 81.709, A4 122.562, A5 -49.215, A6 0.000, E1 2064.07, E2 0, E3 0, E4 0, E5 0, E6 0} C_DIS
   SPTP {A1 6.877, A2 -68.755, A3 82.859, A4 122.310, A5 -47.327, A6 0.000, E1 2066.52, E2 0, E3 0, E4 0, E5 0, E6 0} C_DIS
   SPTP {A1 6.592, A2 -69.340, A3 83.988, A4 121.933, A5 -45.463, A6 0.000, E1 2069.08, E2 0, E3 0, E4 0, E5 0, E6 0} C_DIS
   SPTP {A1 6.317, A2 -69.889, A3 85.097, A4 121.416, A5 -43.626, A6 0.000, E1 2071.77, E2 0, E3 0, E4 0, E5 0, E6 0} C_DIS
   SPTP {A1 6.059, A2 -70.426, A3 86.304, A4 120.438, A5 -41.690, A6 0.000, E1 2074.97, E2 0, E3 0, E4 0, E5 0, E6 0} C_DIS
   SPTP {A1 5.819, A2 -71.023, A3 88.098, A4 117.484, A5 -39.121, A6 0.000, E1 2080.46, E2 0, E3 0, E4 0, E5 0, E6 0} C_DIS
   SPTP {A1 5.593, A2 -71.522, A3 89.806, A4 113.965, A5 -36.737, A6 0.000, E1 2086.48, E2 0, E3 0, E4 0, E5 0, E6 0} C_DIS
   SPTP {A1 5.379, A2 -71.926, A3 91.427, A4 109.828, A5 -34.577, A6 0.000, E1 2093.08, E2 0, E3 0, E4 0, E5 0, E6 0} C_DIS
   SPTP {A1 5.176, A2 -72.232, A3 92.959, A4 105.035, A5 -32.690, A6 0.000, E1 2100.29, E2 0, E3 0, E4 0, E5 0, E6 0} C_DIS
   SPTP {A1 4.988, A2 -72.438, A3 94.394, A4 99.592, A5 -31.143, A6 0.000, E1 2108.13, E2 0, E3 0, E4 0, E5 0, E6 0} C_DIS
   SPTP {A1 4.815, A2 -72.524, A3 95.823, A4 92.947, A5 -30.024, A6 0.000, E1 2117.13, E2 0, E3 0, E4 0, E5 0, E6 0} C_DIS
   SPTP {A1 4.651, A2 -72.464, A3 97.234, A4 85.128, A5 -29.494, A6 0.000, E1 2127.24, E2 0, E3 0, E4 0, E5 0, E6 0} C_DIS
   SPTP {A1 4.493, A2 -72.273, A3 98.499, A4 77.187, A5 -29.603, A6 0.000, E1 2137.45, E2 0, E3 0, E4 0, E5 0, E6 0} C_DIS
   SPTP {A1 4.343, A2 -71.952, A3 99.613, A4 69.494, A5 -30.335, A6 0.000, E1 2147.4, E2 0, E3 0, E4 0, E5 0, E6 0} C_DIS
   SPTP {A1 4.203, A2 -71.502, A3 100.572, A4 62.369, A5 -31.644, A6 0.000, E1 2156.76, E2 0, E3 0, E4 0, E5 0, E6 0} C_DIS
   SPTP {A1 4.077, A2 -70.927, A3 101.368, A4 56.027, A5 -33.457, A6 0.000, E1 2165.35, E2 0, E3 0, E4 0, E5 0, E6 0} C_DIS
   SPTP {A1 3.965, A2 -70.231, A3 102.000, A4 50.536, A5 -35.674, A6 0.000, E1 2173.1, E2 0, E3 0, E4 0, E5 0, E6 0} C_DIS
   SPTP {A1 3.866, A2 -69.423, A3 102.466, A4 45.868, A5 -38.201, A6 0.000, E1 2180.03, E2 0, E3 0, E4 0, E5 0, E6 0} C_DIS
   SPTP {A1 3.784, A2 -68.507, A3 102.765, A4 41.965, A5 -40.961, A6 0.000, E1 2186.22, E2 0, E3 0, E4 0, E5 0, E6 0} C_DIS
   SPTP {A1 3.722, A2 -67.517, A3 102.895, A4 38.799, A5 -43.819, A6 0.000, E1 2191.67, E2 0, E3 0, E4 0, E5 0, E6 0} C_DIS
   SPTP {A1 3.671, A2 -66.785, A3 102.947, A4 36.771, A5 -45.935, A6 0.000, E1 2195.71, E2 0, E3 0, E4 0, E5 0, E6 0} C_DIS
   SPTP {A1 3.641, A2 -66.005, A3 102.903, A4 35.064, A5 -48.103, A6 0.000, E1 2199.46, E2 0, E3 0, E4 0, E5 0, E6 0} C_DIS
   SPTP {A1 3.631, A2 -65.182, A3 102.768, A4 33.640, A5 -50.301, A6 0.000, E1 2202.96, E2 0, E3 0, E4 0, E5 0, E6 0} C_DIS
   SPTP {A1 3.639, A2 -64.319, A3 102.540, A4 32.470, A5 -52.513, A6 0.000, E1 2206.25, E2 0, E3 0, E4 0, E5 0, E6 0} C_DIS
   SPTP {A1 3.667, A2 -63.420, A3 102.221, A4 31.531, A5 -54.726, A6 0.000, E1 2209.33, E2 0, E3 0, E4 0, E5 0, E6 0} C_DIS
   SPTP {A1 3.714, A2 -62.488, A3 101.812, A4 30.801, A5 -56.927, A6 0.000, E1 2212.25, E2 0, E3 0, E4 0, E5 0, E6 0} C_DIS
   SPTP {A1 3.805, A2 -61.792, A3 101.450, A4 30.521, A5 -58.551, A6 0.000, E1 2214.72, E2 0, E3 0, E4 0, E5 0, E6 0} C_DIS
   SPTP {A1 3.932, A2 -61.284, A3 101.142, A4 30.561, A5 -59.736, A6 0.000, E1 2216.88, E2 0, E3 0, E4 0, E5 0, E6 0} C_DIS
   SPTP {A1 4.076, A2 -60.767, A3 100.794, A4 30.708, A5 -60.909, A6 0.000, E1 2218.96, E2 0, E3 0, E4 0, E5 0, E6 0} C_DIS
   SPTP {A1 4.235, A2 -60.242, A3 100.407, A4 30.952, A5 -62.068, A6 0.000, E1 2220.97, E2 0, E3 0, E4 0, E5 0, E6 0} C_DIS
   SPTP {A1 4.405, A2 -59.711, A3 99.984, A4 31.271, A5 -63.206, A6 0.000, E1 2222.93, E2 0, E3 0, E4 0, E5 0, E6 0} C_DIS
   SPTP {A1 4.586, A2 -59.173, A3 99.526, A4 31.666, A5 -64.323, A6 0.000, E1 2224.83, E2 0, E3 0, E4 0, E5 0, E6 0} C_DIS
   SPTP {A1 4.776, A2 -58.631, A3 99.031, A4 32.131, A5 -65.419, A6 0.000, E1 2226.69, E2 0, E3 0, E4 0, E5 0, E6 0} C_DIS
   SPTP {A1 4.974, A2 -58.084, A3 98.503, A4 32.655, A5 -66.490, A6 0.000, E1 2228.51, E2 0, E3 0, E4 0, E5 0, E6 0} C_DIS
   SPTP {A1 5.230, A2 -57.828, A3 98.128, A4 33.534, A5 -66.981, A6 0.000, E1 2230.03, E2 0, E3 0, E4 0, E5 0, E6 0} C_DIS
   SPTP {A1 5.508, A2 -57.657, A3 97.782, A4 34.555, A5 -67.294, A6 0.000, E1 2231.43, E2 0, E3 0, E4 0, E5 0, E6 0} C_DIS
   SPTP {A1 5.790, A2 -57.484, A3 97.414, A4 35.615, A5 -67.595, A6 0.000, E1 2232.8, E2 0, E3 0, E4 0, E5 0, E6 0} C_DIS
   SPTP {A1 6.073, A2 -57.308, A3 97.022, A4 36.710, A5 -67.884, A6 0.000, E1 2234.14, E2 0, E3 0, E4 0, E5 0, E6 0} C_DIS
   SPTP {A1 6.359, A2 -57.130, A3 96.607, A4 37.838, A5 -68.163, A6 0.000, E1 2235.44, E2 0, E3 0, E4 0, E5 0, E6 0} C_DIS
   SPTP {A1 6.644, A2 -56.949, A3 96.170, A4 38.993, A5 -68.432, A6 0.000, E1 2236.72, E2 0, E3 0, E4 0, E5 0, E6 0} C_DIS
   SPTP {A1 6.927, A2 -56.765, A3 95.710, A4 40.170, A5 -68.690, A6 0.000, E1 2237.97, E2 0, E3 0, E4 0, E5 0, E6 0} C_DIS
   SPTP {A1 7.209, A2 -56.579, A3 95.230, A4 41.365, A5 -68.939, A6 0.000, E1 2239.2, E2 0, E3 0, E4 0, E5 0, E6 0} C_DIS
   SPTP {A1 7.486, A2 -56.392, A3 94.730, A4 42.575, A5 -69.176, A6 0.000, E1 2240.41, E2 0, E3 0, E4 0, E5 0, E6 0} C_DIS
   SPTP {A1 7.759, A2 -56.203, A3 94.213, A4 43.795, A5 -69.403, A6 0.000, E1 2241.61, E2 0, E3 0, E4 0, E5 0, E6 0} C_DIS
   SPTP {A1 8.026, A2 -56.015, A3 93.679, A4 45.019, A5 -69.617, A6 0.000, E1 2242.79, E2 0, E3 0, E4 0, E5 0, E6 0} C_DIS
   SPTP {A1 8.287, A2 -55.831, A3 93.134, A4 46.251, A5 -69.814, A6 0.000, E1 2243.96, E2 0, E3 0, E4 0, E5 0, E6 0} C_DIS
   SPTP {A1 8.553, A2 -55.767, A3 92.660, A4 47.603, A5 -69.800, A6 0.000, E1 2244.93, E2 0, E3 0, E4 0, E5 0, E6 0} C_DIS
   SPTP {A1 8.813, A2 -55.700, A3 92.171, A4 48.960, A5 -69.782, A6 0.000, E1 2245.88, E2 0, E3 0, E4 0, E5 0, E6 0} C_DIS
   SPTP {A1 9.064, A2 -55.632, A3 91.666, A4 50.318, A5 -69.760, A6 0.000, E1 2246.83, E2 0, E3 0, E4 0, E5 0, E6 0} C_DIS
   SPTP {A1 9.307, A2 -55.563, A3 91.149, A4 51.674, A5 -69.733, A6 0.000, E1 2247.76, E2 0, E3 0, E4 0, E5 0, E6 0} C_DIS
   SPTP {A1 9.540, A2 -55.494, A3 90.622, A4 53.026, A5 -69.700, A6 0.000, E1 2248.68, E2 0, E3 0, E4 0, E5 0, E6 0} C_DIS
   SPTP {A1 9.765, A2 -55.425, A3 90.085, A4 54.374, A5 -69.663, A6 0.000, E1 2249.6, E2 0, E3 0, E4 0, E5 0, E6 0} C_DIS
   SPTP {A1 9.979, A2 -55.359, A3 89.541, A4 55.711, A5 -69.617, A6 0.000, E1 2250.52, E2 0, E3 0, E4 0, E5 0, E6 0} C_DIS
   SPTP {A1 10.183, A2 -55.295, A3 88.993, A4 57.039, A5 -69.566, A6 0.000, E1 2251.44, E2 0, E3 0, E4 0, E5 0, E6 0} C_DIS
   SPTP {A1 10.376, A2 -55.234, A3 88.443, A4 58.355, A5 -69.506, A6 0.000, E1 2252.35, E2 0, E3 0, E4 0, E5 0, E6 0} C_DIS
   SPTP {A1 10.559, A2 -55.178, A3 87.893, A4 59.657, A5 -69.437, A6 0.000, E1 2253.27, E2 0, E3 0, E4 0, E5 0, E6 0} C_DIS
   SPTP {A1 10.720, A2 -55.130, A3 87.373, A4 60.885, A5 -69.378, A6 0.000, E1 2254.17, E2 0, E3 0, E4 0, E5 0, E6 0} C_DIS
   SPTP {A1 10.867, A2 -55.089, A3 86.865, A4 62.082, A5 -69.313, A6 0.000, E1 2255.07, E2 0, E3 0, E4 0, E5 0, E6 0} C_DIS
   SPTP {A1 10.978, A2 -55.057, A3 86.432, A4 63.115, A5 -69.287, A6 0.000, E1 2255.93, E2 0, E3 0, E4 0, E5 0, E6 0} C_DIS
   SPTP {A1 11.081, A2 -55.034, A3 86.009, A4 64.131, A5 -69.247, A6 0.000, E1 2256.8, E2 0, E3 0, E4 0, E5 0, E6 0} C_DIS
   SPTP {A1 11.175, A2 -55.020, A3 85.598, A4 65.129, A5 -69.194, A6 0.000, E1 2257.68, E2 0, E3 0, E4 0, E5 0, E6 0} C_DIS
   SPTP {A1 11.261, A2 -55.018, A3 85.202, A4 66.107, A5 -69.123, A6 0.000, E1 2258.57, E2 0, E3 0, E4 0, E5 0, E6 0} C_DIS
   SPTP {A1 11.339, A2 -55.027, A3 84.821, A4 67.066, A5 -69.035, A6 0.000, E1 2259.48, E2 0, E3 0, E4 0, E5 0, E6 0} C_DIS
   SPTP {A1 11.408, A2 -55.048, A3 84.458, A4 68.005, A5 -68.930, A6 0.000, E1 2260.4, E2 0, E3 0, E4 0, E5 0, E6 0} C_DIS
   SPTP {A1 11.469, A2 -55.084, A3 84.116, A4 68.922, A5 -68.802, A6 0.000, E1 2261.34, E2 0, E3 0, E4 0, E5 0, E6 0} C_DIS
   SPTP {A1 11.522, A2 -55.134, A3 83.795, A4 69.819, A5 -68.653, A6 0.000, E1 2262.29, E2 0, E3 0, E4 0, E5 0, E6 0} C_DIS
   SPTP {A1 11.567, A2 -55.198, A3 83.495, A4 70.695, A5 -68.484, A6 0.000, E1 2263.26, E2 0, E3 0, E4 0, E5 0, E6 0} C_DIS
   SPTP {A1 11.604, A2 -55.277, A3 83.219, A4 71.551, A5 -68.291, A6 0.000, E1 2264.24, E2 0, E3 0, E4 0, E5 0, E6 0} C_DIS
   SPTP {A1 11.632, A2 -55.373, A3 82.969, A4 72.384, A5 -68.073, A6 0.000, E1 2265.24, E2 0, E3 0, E4 0, E5 0, E6 0} C_DIS
   SPTP {A1 11.653, A2 -55.485, A3 82.744, A4 73.197, A5 -67.831, A6 0.000, E1 2266.26, E2 0, E3 0, E4 0, E5 0, E6 0} C_DIS
   SPTP {A1 11.666, A2 -55.613, A3 82.546, A4 73.989, A5 -67.563, A6 0.000, E1 2267.29, E2 0, E3 0, E4 0, E5 0, E6 0} C_DIS
   SPTP {A1 11.671, A2 -55.758, A3 82.376, A4 74.760, A5 -67.267, A6 0.000, E1 2268.34, E2 0, E3 0, E4 0, E5 0, E6 0} C_DIS
   SPTP {A1 11.668, A2 -55.922, A3 82.235, A4 75.508, A5 -66.943, A6 0.000, E1 2269.4, E2 0, E3 0, E4 0, E5 0, E6 0} C_DIS
   SPTP {A1 11.657, A2 -56.103, A3 82.124, A4 76.235, A5 -66.589, A6 0.000, E1 2270.48, E2 0, E3 0, E4 0, E5 0, E6 0} C_DIS
   SPTP {A1 11.638, A2 -56.304, A3 82.044, A4 76.944, A5 -66.206, A6 0.000, E1 2271.56, E2 0, E3 0, E4 0, E5 0, E6 0} C_DIS
   SPTP {A1 11.603, A2 -56.573, A3 82.052, A4 77.666, A5 -65.761, A6 0.000, E1 2272.35, E2 0, E3 0, E4 0, E5 0, E6 0} C_DIS
   SPTP {A1 11.560, A2 -56.854, A3 82.080, A4 78.376, A5 -65.295, A6 0.000, E1 2273.15, E2 0, E3 0, E4 0, E5 0, E6 0} C_DIS
   SPTP {A1 11.511, A2 -57.146, A3 82.127, A4 79.073, A5 -64.806, A6 0.000, E1 2273.95, E2 0, E3 0, E4 0, E5 0, E6 0} C_DIS
   SPTP {A1 11.455, A2 -57.452, A3 82.197, A4 79.755, A5 -64.292, A6 0.000, E1 2274.76, E2 0, E3 0, E4 0, E5 0, E6 0} C_DIS
   SPTP {A1 11.391, A2 -57.769, A3 82.287, A4 80.424, A5 -63.753, A6 0.000, E1 2275.58, E2 0, E3 0, E4 0, E5 0, E6 0} C_DIS
   SPTP {A1 11.319, A2 -58.100, A3 82.399, A4 81.078, A5 -63.188, A6 0.000, E1 2276.4, E2 0, E3 0, E4 0, E5 0, E6 0} C_DIS
   SPTP {A1 11.240, A2 -58.444, A3 82.533, A4 81.716, A5 -62.595, A6 0.000, E1 2277.23, E2 0, E3 0, E4 0, E5 0, E6 0} C_DIS
   SPTP {A1 11.152, A2 -58.799, A3 82.689, A4 82.341, A5 -61.974, A6 0.000, E1 2278.06, E2 0, E3 0, E4 0, E5 0, E6 0} C_DIS
   SPTP {A1 11.057, A2 -59.167, A3 82.865, A4 82.952, A5 -61.326, A6 0.000, E1 2278.9, E2 0, E3 0, E4 0, E5 0, E6 0} C_DIS
   SPTP {A1 10.953, A2 -59.547, A3 83.063, A4 83.548, A5 -60.648, A6 0.000, E1 2279.74, E2 0, E3 0, E4 0, E5 0, E6 0} C_DIS
   SPTP {A1 10.841, A2 -59.938, A3 83.281, A4 84.130, A5 -59.941, A6 0.000, E1 2280.59, E2 0, E3 0, E4 0, E5 0, E6 0} C_DIS
   SPTP {A1 10.721, A2 -60.353, A3 83.498, A4 84.797, A5 -59.180, A6 0.000, E1 2281.32, E2 0, E3 0, E4 0, E5 0, E6 0} C_DIS
   SPTP {A1 10.599, A2 -60.826, A3 83.636, A4 85.894, A5 -58.291, A6 0.000, E1 2281.56, E2 0, E3 0, E4 0, E5 0, E6 0} C_DIS
   SPTP {A1 10.466, A2 -61.301, A3 83.777, A4 87.005, A5 -57.390, A6 0.000, E1 2281.78, E2 0, E3 0, E4 0, E5 0, E6 0} C_DIS
   SPTP {A1 10.321, A2 -61.778, A3 83.925, A4 88.127, A5 -56.472, A6 0.000, E1 2281.96, E2 0, E3 0, E4 0, E5 0, E6 0} C_DIS
   SPTP {A1 10.164, A2 -62.257, A3 84.079, A4 89.263, A5 -55.541, A6 0.000, E1 2282.13, E2 0, E3 0, E4 0, E5 0, E6 0} C_DIS
   SPTP {A1 9.996, A2 -62.736, A3 84.236, A4 90.417, A5 -54.599, A6 0.000, E1 2282.26, E2 0, E3 0, E4 0, E5 0, E6 0} C_DIS
   SPTP {A1 9.816, A2 -63.215, A3 84.396, A4 91.590, A5 -53.646, A6 0.000, E1 2282.36, E2 0, E3 0, E4 0, E5 0, E6 0} C_DIS
   SPTP {A1 9.624, A2 -63.693, A3 84.559, A4 92.784, A5 -52.681, A6 0.000, E1 2282.42, E2 0, E3 0, E4 0, E5 0, E6 0} C_DIS
   SPTP {A1 9.420, A2 -64.171, A3 84.726, A4 94.001, A5 -51.706, A6 0.000, E1 2282.45, E2 0, E3 0, E4 0, E5 0, E6 0} C_DIS
   SPTP {A1 9.204, A2 -64.647, A3 84.895, A4 95.245, A5 -50.721, A6 0.000, E1 2282.45, E2 0, E3 0, E4 0, E5 0, E6 0} C_DIS
   SPTP {A1 8.975, A2 -65.120, A3 85.067, A4 96.518, A5 -49.727, A6 0.000, E1 2282.4, E2 0, E3 0, E4 0, E5 0, E6 0} C_DIS
   SPTP {A1 8.735, A2 -65.591, A3 85.239, A4 97.823, A5 -48.725, A6 0.000, E1 2282.3, E2 0, E3 0, E4 0, E5 0, E6 0} C_DIS
   SPTP {A1 8.483, A2 -66.059, A3 85.413, A4 99.163, A5 -47.717, A6 0.000, E1 2282.16, E2 0, E3 0, E4 0, E5 0, E6 0} C_DIS
   SPTP {A1 8.218, A2 -66.522, A3 85.587, A4 100.543, A5 -46.705, A6 0.000, E1 2281.97, E2 0, E3 0, E4 0, E5 0, E6 0} C_DIS
   SPTP {A1 7.942, A2 -66.980, A3 85.760, A4 101.966, A5 -45.691, A6 0.000, E1 2281.73, E2 0, E3 0, E4 0, E5 0, E6 0} C_DIS
   SPTP {A1 7.648, A2 -67.436, A3 85.886, A4 103.630, A5 -44.647, A6 0.000, E1 2281.33, E2 0, E3 0, E4 0, E5 0, E6 0} C_DIS
   SPTP {A1 7.332, A2 -67.891, A3 85.945, A4 105.640, A5 -43.566, A6 0.000, E1 2280.71, E2 0, E3 0, E4 0, E5 0, E6 0} C_DIS
   SPTP {A1 7.001, A2 -68.334, A3 86.000, A4 107.728, A5 -42.505, A6 0.000, E1 2280, E2 0, E3 0, E4 0, E5 0, E6 0} C_DIS
   SPTP {A1 6.655, A2 -68.767, A3 86.052, A4 109.899, A5 -41.463, A6 0.000, E1 2279.2, E2 0, E3 0, E4 0, E5 0, E6 0} C_DIS
   SPTP {A1 6.296, A2 -69.187, A3 86.101, A4 112.157, A5 -40.449, A6 0.000, E1 2278.31, E2 0, E3 0, E4 0, E5 0, E6 0} C_DIS
   SPTP {A1 5.922, A2 -69.596, A3 86.146, A4 114.508, A5 -39.461, A6 0.000, E1 2277.32, E2 0, E3 0, E4 0, E5 0, E6 0} C_DIS
   SPTP {A1 5.536, A2 -69.990, A3 86.185, A4 116.954, A5 -38.513, A6 0.000, E1 2276.22, E2 0, E3 0, E4 0, E5 0, E6 0} C_DIS
   SPTP {A1 5.139, A2 -70.368, A3 86.218, A4 119.497, A5 -37.610, A6 0.000, E1 2275.04, E2 0, E3 0, E4 0, E5 0, E6 0} C_DIS
   SPTP {A1 4.734, A2 -70.731, A3 86.244, A4 122.136, A5 -36.760, A6 0.000, E1 2273.75, E2 0, E3 0, E4 0, E5 0, E6 0} C_DIS
   SPTP {A1 4.319, A2 -71.077, A3 86.264, A4 124.868, A5 -35.968, A6 0.000, E1 2272.38, E2 0, E3 0, E4 0, E5 0, E6 0} C_DIS
   SPTP {A1 3.899, A2 -71.406, A3 86.276, A4 127.687, A5 -35.240, A6 0.000, E1 2270.92, E2 0, E3 0, E4 0, E5 0, E6 0} C_DIS
   SPTP {A1 3.471, A2 -71.719, A3 86.283, A4 130.590, A5 -34.576, A6 0.000, E1 2269.38, E2 0, E3 0, E4 0, E5 0, E6 0} C_DIS
   SPTP {A1 3.039, A2 -72.016, A3 86.285, A4 133.565, A5 -33.982, A6 0.000, E1 2267.78, E2 0, E3 0, E4 0, E5 0, E6 0} C_DIS
   SPTP {A1 2.606, A2 -72.295, A3 86.280, A4 136.594, A5 -33.469, A6 0.000, E1 2266.14, E2 0, E3 0, E4 0, E5 0, E6 0} C_DIS
   SPTP {A1 2.171, A2 -72.647, A3 86.607, A4 138.971, A5 -32.495, A6 0.000, E1 2265.33, E2 0, E3 0, E4 0, E5 0, E6 0} C_DIS
   SPTP {A1 1.736, A2 -73.017, A3 87.052, A4 141.187, A5 -31.366, A6 0.000, E1 2264.73, E2 0, E3 0, E4 0, E5 0, E6 0} C_DIS
   SPTP {A1 1.304, A2 -73.377, A3 87.505, A4 143.483, A5 -30.261, A6 0.000, E1 2264.05, E2 0, E3 0, E4 0, E5 0, E6 0} C_DIS
   SPTP {A1 0.878, A2 -73.724, A3 87.964, A4 145.854, A5 -29.184, A6 0.000, E1 2263.31, E2 0, E3 0, E4 0, E5 0, E6 0} C_DIS
   SPTP {A1 0.463, A2 -74.059, A3 88.428, A4 148.283, A5 -28.144, A6 0.000, E1 2262.52, E2 0, E3 0, E4 0, E5 0, E6 0} C_DIS
   SPTP {A1 0.063, A2 -74.383, A3 88.898, A4 150.749, A5 -27.145, A6 0.000, E1 2261.72, E2 0, E3 0, E4 0, E5 0, E6 0} C_DIS
   SPTP {A1 -0.318, A2 -74.694, A3 89.374, A4 153.229, A5 -26.188, A6 0.000, E1 2260.93, E2 0, E3 0, E4 0, E5 0, E6 0} C_DIS
   SPTP {A1 -0.670, A2 -75.079, A3 90.225, A4 154.892, A5 -24.577, A6 0.000, E1 2260.97, E2 0, E3 0, E4 0, E5 0, E6 0} C_DIS
   SPTP {A1 -0.990, A2 -75.514, A3 91.416, A4 155.704, A5 -22.315, A6 0.000, E1 2261.88, E2 0, E3 0, E4 0, E5 0, E6 0} C_DIS
   SPTP {A1 -1.277, A2 -75.913, A3 92.588, A4 156.366, A5 -20.060, A6 0.000, E1 2262.95, E2 0, E3 0, E4 0, E5 0, E6 0} C_DIS
   SPTP {A1 -1.529, A2 -76.277, A3 93.742, A4 156.795, A5 -17.811, A6 0.000, E1 2264.27, E2 0, E3 0, E4 0, E5 0, E6 0} C_DIS
   SPTP {A1 -1.734, A2 -76.605, A3 94.876, A4 156.786, A5 -15.583, A6 0.000, E1 2266.05, E2 0, E3 0, E4 0, E5 0, E6 0} C_DIS
   SPTP {A1 -1.889, A2 -76.924, A3 96.376, A4 154.167, A5 -12.497, A6 0.000, E1 2270.45, E2 0, E3 0, E4 0, E5 0, E6 0} C_DIS
   SPTP {A1 -1.995, A2 -77.169, A3 98.183, A4 145.295, A5 -8.671, A6 0.000, E1 2281.06, E2 0, E3 0, E4 0, E5 0, E6 0} C_DIS
   SPTP {A1 -2.050, A2 -77.285, A3 99.872, A4 122.916, A5 -5.483, A6 0.000, E1 2305.19, E2 0, E3 0, E4 0, E5 0, E6 0} C_DIS
   SPTP {A1 -2.051, A2 -77.272, A3 101.437, A4 74.993, A5 -4.605, A6 0.000, E1 2354.87, E2 0, E3 0, E4 0, E5 0, E6 0} C_DIS
   SPTP {A1 -1.998, A2 -77.121, A3 102.887, A4 39.468, A5 -7.051, A6 0.000, E1 2392.18, E2 0, E3 0, E4 0, E5 0, E6 0} C_DIS
   SPTP {A1 -1.911, A2 -76.538, A3 104.701, A4 21.441, A5 -12.806, A6 0.000, E1 2412, E2 0, E3 0, E4 0, E5 0, E6 0} C_DIS
   SPTP {A1 -1.782, A2 -75.655, A3 106.171, A4 15.430, A5 -19.048, A6 0.000, E1 2419.81, E2 0, E3 0, E4 0, E5 0, E6 0} C_DIS
   SPTP {A1 -1.624, A2 -74.483, A3 107.286, A4 12.782, A5 -25.371, A6 0.000, E1 2424.24, E2 0, E3 0, E4 0, E5 0, E6 0} C_DIS
   SPTP {A1 -1.443, A2 -72.662, A3 108.096, A4 10.989, A5 -32.964, A6 0.000, E1 2428.02, E2 0, E3 0, E4 0, E5 0, E6 0} C_DIS
   SPTP {A1 -1.248, A2 -70.202, A3 108.323, A4 9.921, A5 -41.220, A6 0.000, E1 2431.19, E2 0, E3 0, E4 0, E5 0, E6 0} C_DIS
   SPTP {A1 -1.050, A2 -67.371, A3 107.856, A4 9.442, A5 -49.186, A6 0.000, E1 2433.8, E2 0, E3 0, E4 0, E5 0, E6 0} C_DIS
   SPTP {A1 -0.859, A2 -64.248, A3 106.701, A4 9.277, A5 -56.772, A6 0.000, E1 2436.12, E2 0, E3 0, E4 0, E5 0, E6 0} C_DIS
   SPTP {A1 -0.563, A2 -61.304, A3 105.107, A4 9.646, A5 -63.116, A6 0.000, E1 2438.41, E2 0, E3 0, E4 0, E5 0, E6 0} C_DIS
   SPTP {A1 -0.142, A2 -58.644, A3 103.274, A4 10.510, A5 -68.315, A6 0.000, E1 2440.74, E2 0, E3 0, E4 0, E5 0, E6 0} C_DIS
   SPTP {A1 0.295, A2 -55.938, A3 101.051, A4 11.517, A5 -73.149, A6 0.000, E1 2443.04, E2 0, E3 0, E4 0, E5 0, E6 0} C_DIS
   SPTP {A1 0.748, A2 -53.210, A3 98.454, A4 12.681, A5 -77.608, A6 0.000, E1 2445.29, E2 0, E3 0, E4 0, E5 0, E6 0} C_DIS
   SPTP {A1 1.207, A2 -50.480, A3 95.504, A4 13.960, A5 -81.685, A6 0.000, E1 2447.52, E2 0, E3 0, E4 0, E5 0, E6 0} C_DIS
   SPTP {A1 1.669, A2 -47.759, A3 92.215, A4 15.353, A5 -85.383, A6 0.000, E1 2449.74, E2 0, E3 0, E4 0, E5 0, E6 0} C_DIS
   SPTP {A1 2.137, A2 -45.047, A3 88.589, A4 16.880, A5 -88.709, A6 0.000, E1 2451.91, E2 0, E3 0, E4 0, E5 0, E6 0} C_DIS
   SPTP {A1 2.607, A2 -42.337, A3 84.624, A4 18.524, A5 -91.674, A6 0.000, E1 2454.02, E2 0, E3 0, E4 0, E5 0, E6 0} C_DIS
   SPTP {A1 3.074, A2 -39.618, A3 80.312, A4 20.276, A5 -94.285, A6 0.000, E1 2456.06, E2 0, E3 0, E4 0, E5 0, E6 0} C_DIS
   SPTP {A1 3.536, A2 -36.861, A3 75.620, A4 22.127, A5 -96.551, A6 0.000, E1 2457.99, E2 0, E3 0, E4 0, E5 0, E6 0} C_DIS
   SPTP {A1 4.023, A2 -34.845, A3 71.855, A4 24.115, A5 -97.924, A6 0.000, E1 2459.67, E2 0, E3 0, E4 0, E5 0, E6 0} C_DIS
   SPTP {A1 4.589, A2 -34.730, A3 71.122, A4 26.315, A5 -97.838, A6 0.000, E1 2460.9, E2 0, E3 0, E4 0, E5 0, E6 0} C_DIS
   SPTP {A1 5.147, A2 -34.594, A3 70.299, A4 28.578, A5 -97.719, A6 0.000, E1 2461.97, E2 0, E3 0, E4 0, E5 0, E6 0} C_DIS
   SPTP {A1 5.693, A2 -34.432, A3 69.378, A4 30.888, A5 -97.576, A6 0.000, E1 2462.9, E2 0, E3 0, E4 0, E5 0, E6 0} C_DIS
   SPTP {A1 6.194, A2 -34.789, A3 69.341, A4 33.082, A5 -97.095, A6 0.000, E1 2463.49, E2 0, E3 0, E4 0, E5 0, E6 0} C_DIS
   SPTP {A1 6.669, A2 -35.415, A3 69.741, A4 35.231, A5 -96.416, A6 0.000, E1 2463.82, E2 0, E3 0, E4 0, E5 0, E6 0} C_DIS
   SPTP {A1 7.057, A2 -35.900, A3 69.981, A4 37.039, A5 -95.846, A6 0.000, E1 2464.01, E2 0, E3 0, E4 0, E5 0, E6 0} C_DIS
   SPTP {A1 7.438, A2 -36.359, A3 70.148, A4 38.862, A5 -95.271, A6 0.000, E1 2464.13, E2 0, E3 0, E4 0, E5 0, E6 0} C_DIS
   SPTP {A1 7.439, A2 -36.344, A3 70.130, A4 38.875, A5 -95.282, A6 0.000, E1 2464.11, E2 0, E3 0, E4 0, E5 0, E6 0} C_DIS
   SPTP {A1 7.886, A2 -36.867, A3 70.247, A4 41.078, A5 -94.585, A6 0.000, E1 2464.19, E2 0, E3 0, E4 0, E5 0, E6 0} C_DIS
   SPTP {A1 8.290, A2 -37.633, A3 70.781, A4 43.148, A5 -93.720, A6 0.000, E1 2464.03, E2 0, E3 0, E4 0, E5 0, E6 0} C_DIS
   SPTP {A1 8.654, A2 -38.641, A3 71.718, A4 45.096, A5 -92.670, A6 0.000, E1 2463.59, E2 0, E3 0, E4 0, E5 0, E6 0} C_DIS
   SPTP {A1 9.010, A2 -39.618, A3 72.553, A4 47.058, A5 -91.599, A6 0.000, E1 2463.09, E2 0, E3 0, E4 0, E5 0, E6 0} C_DIS
   SPTP {A1 9.359, A2 -40.564, A3 73.289, A4 49.041, A5 -90.512, A6 0.000, E1 2462.52, E2 0, E3 0, E4 0, E5 0, E6 0} C_DIS
   SPTP {A1 9.696, A2 -41.485, A3 73.941, A4 51.034, A5 -89.412, A6 0.000, E1 2461.9, E2 0, E3 0, E4 0, E5 0, E6 0} C_DIS
   SPTP {A1 10.022, A2 -42.388, A3 74.523, A4 53.034, A5 -88.296, A6 0.000, E1 2461.23, E2 0, E3 0, E4 0, E5 0, E6 0} C_DIS
   SPTP {A1 10.334, A2 -43.280, A3 75.049, A4 55.036, A5 -87.162, A6 0.000, E1 2460.52, E2 0, E3 0, E4 0, E5 0, E6 0} C_DIS
   SPTP {A1 10.630, A2 -44.163, A3 75.522, A4 57.039, A5 -86.012, A6 0.000, E1 2459.77, E2 0, E3 0, E4 0, E5 0, E6 0} C_DIS
   SPTP {A1 10.887, A2 -45.147, A3 76.157, A4 58.947, A5 -84.780, A6 0.000, E1 2458.81, E2 0, E3 0, E4 0, E5 0, E6 0} C_DIS
   SPTP {A1 11.119, A2 -46.171, A3 76.827, A4 60.821, A5 -83.495, A6 0.000, E1 2457.72, E2 0, E3 0, E4 0, E5 0, E6 0} C_DIS
   SPTP {A1 11.336, A2 -47.164, A3 77.408, A4 62.733, A5 -82.219, A6 0.000, E1 2456.55, E2 0, E3 0, E4 0, E5 0, E6 0} C_DIS
   SPTP {A1 11.535, A2 -48.153, A3 77.944, A4 64.655, A5 -80.923, A6 0.000, E1 2455.33, E2 0, E3 0, E4 0, E5 0, E6 0} C_DIS
   SPTP {A1 11.716, A2 -49.122, A3 78.415, A4 66.607, A5 -79.630, A6 0.000, E1 2454.03, E2 0, E3 0, E4 0, E5 0, E6 0} C_DIS
   SPTP {A1 11.876, A2 -50.085, A3 78.841, A4 68.577, A5 -78.325, A6 0.000, E1 2452.68, E2 0, E3 0, E4 0, E5 0, E6 0} C_DIS
   SPTP {A1 12.014, A2 -51.032, A3 79.212, A4 70.577, A5 -77.023, A6 0.000, E1 2451.26, E2 0, E3 0, E4 0, E5 0, E6 0} C_DIS
   SPTP {A1 12.130, A2 -51.962, A3 79.528, A4 72.612, A5 -75.730, A6 0.000, E1 2449.75, E2 0, E3 0, E4 0, E5 0, E6 0} C_DIS
   SPTP {A1 12.221, A2 -52.879, A3 79.796, A4 74.681, A5 -74.442, A6 0.000, E1 2448.18, E2 0, E3 0, E4 0, E5 0, E6 0} C_DIS
   SPTP {A1 12.289, A2 -53.768, A3 79.998, A4 76.800, A5 -73.183, A6 0.000, E1 2446.51, E2 0, E3 0, E4 0, E5 0, E6 0} C_DIS
   SPTP {A1 12.330, A2 -54.645, A3 80.157, A4 78.959, A5 -71.937, A6 0.000, E1 2444.75, E2 0, E3 0, E4 0, E5 0, E6 0} C_DIS
   SPTP {A1 12.347, A2 -55.484, A3 80.240, A4 81.182, A5 -70.741, A6 0.000, E1 2442.9, E2 0, E3 0, E4 0, E5 0, E6 0} C_DIS
   SPTP {A1 12.336, A2 -56.306, A3 80.278, A4 83.453, A5 -69.570, A6 0.000, E1 2440.95, E2 0, E3 0, E4 0, E5 0, E6 0} C_DIS
   SPTP {A1 12.299, A2 -57.075, A3 80.244, A4 85.751, A5 -68.478, A6 0.000, E1 2438.98, E2 0, E3 0, E4 0, E5 0, E6 0} C_DIS
   SPTP {A1 12.230, A2 -57.762, A3 80.201, A4 87.831, A5 -67.466, A6 0.000, E1 2437.48, E2 0, E3 0, E4 0, E5 0, E6 0} C_DIS
   SPTP {A1 12.138, A2 -58.424, A3 80.128, A4 89.932, A5 -66.491, A6 0.000, E1 2435.96, E2 0, E3 0, E4 0, E5 0, E6 0} C_DIS
   SPTP {A1 12.022, A2 -59.068, A3 80.025, A4 92.079, A5 -65.547, A6 0.000, E1 2434.36, E2 0, E3 0, E4 0, E5 0, E6 0} C_DIS
   SPTP {A1 11.881, A2 -59.690, A3 79.887, A4 94.277, A5 -64.645, A6 0.000, E1 2432.69, E2 0, E3 0, E4 0, E5 0, E6 0} C_DIS
   SPTP {A1 11.717, A2 -60.285, A3 79.708, A4 96.531, A5 -63.797, A6 0.000, E1 2430.94, E2 0, E3 0, E4 0, E5 0, E6 0} C_DIS
   SPTP {A1 11.530, A2 -60.852, A3 79.487, A4 98.840, A5 -63.008, A6 0.000, E1 2429.1, E2 0, E3 0, E4 0, E5 0, E6 0} C_DIS
   SPTP {A1 11.322, A2 -61.380, A3 79.212, A4 101.211, A5 -62.298, A6 0.000, E1 2427.19, E2 0, E3 0, E4 0, E5 0, E6 0} C_DIS
   SPTP {A1 11.094, A2 -61.869, A3 78.898, A4 103.601, A5 -61.667, A6 0.000, E1 2425.28, E2 0, E3 0, E4 0, E5 0, E6 0} C_DIS
   SPTP {A1 10.849, A2 -62.367, A3 78.846, A4 105.439, A5 -60.860, A6 0.000, E1 2424.45, E2 0, E3 0, E4 0, E5 0, E6 0} C_DIS
   SPTP {A1 10.586, A2 -62.853, A3 78.785, A4 107.317, A5 -60.075, A6 0.000, E1 2423.57, E2 0, E3 0, E4 0, E5 0, E6 0} C_DIS
   SPTP {A1 10.308, A2 -63.324, A3 78.710, A4 109.237, A5 -59.322, A6 0.000, E1 2422.64, E2 0, E3 0, E4 0, E5 0, E6 0} C_DIS
   SPTP {A1 10.016, A2 -63.771, A3 78.613, A4 111.200, A5 -58.618, A6 0.000, E1 2421.67, E2 0, E3 0, E4 0, E5 0, E6 0} C_DIS
   SPTP {A1 9.713, A2 -64.191, A3 78.486, A4 113.207, A5 -57.977, A6 0.000, E1 2420.65, E2 0, E3 0, E4 0, E5 0, E6 0} C_DIS
   SPTP {A1 9.401, A2 -64.580, A3 78.324, A4 115.255, A5 -57.409, A6 0.000, E1 2419.6, E2 0, E3 0, E4 0, E5 0, E6 0} C_DIS
   SPTP {A1 9.085, A2 -65.022, A3 78.426, A4 116.891, A5 -56.607, A6 0.000, E1 2419.26, E2 0, E3 0, E4 0, E5 0, E6 0} C_DIS
   SPTP {A1 8.763, A2 -65.542, A3 78.844, A4 118.064, A5 -55.487, A6 0.000, E1 2419.71, E2 0, E3 0, E4 0, E5 0, E6 0} C_DIS
   SPTP {A1 8.440, A2 -66.047, A3 79.257, A4 119.249, A5 -54.385, A6 0.000, E1 2420.15, E2 0, E3 0, E4 0, E5 0, E6 0} C_DIS
   SPTP {A1 8.116, A2 -66.534, A3 79.662, A4 120.446, A5 -53.306, A6 0.000, E1 2420.58, E2 0, E3 0, E4 0, E5 0, E6 0} C_DIS
   SPTP {A1 7.794, A2 -67.001, A3 80.056, A4 121.650, A5 -52.258, A6 0.000, E1 2421.02, E2 0, E3 0, E4 0, E5 0, E6 0} C_DIS
   SPTP {A1 7.479, A2 -67.476, A3 80.537, A4 122.697, A5 -51.135, A6 0.000, E1 2421.7, E2 0, E3 0, E4 0, E5 0, E6 0} C_DIS
   SPTP {A1 7.175, A2 -68.128, A3 81.702, A4 122.560, A5 -49.234, A6 0.000, E1 2424.04, E2 0, E3 0, E4 0, E5 0, E6 0} C_DIS
   SPTP {A1 6.879, A2 -68.749, A3 82.853, A4 122.311, A5 -47.343, A6 0.000, E1 2426.48, E2 0, E3 0, E4 0, E5 0, E6 0} C_DIS
   SPTP {A1 6.593, A2 -69.334, A3 83.983, A4 121.937, A5 -45.476, A6 0.000, E1 2429.03, E2 0, E3 0, E4 0, E5 0, E6 0} C_DIS
   SPTP {A1 6.318, A2 -69.885, A3 85.093, A4 121.423, A5 -43.636, A6 0.000, E1 2431.71, E2 0, E3 0, E4 0, E5 0, E6 0} C_DIS
   SPTP {A1 6.057, A2 -70.421, A3 86.285, A4 120.487, A5 -41.714, A6 0.000, E1 2434.86, E2 0, E3 0, E4 0, E5 0, E6 0} C_DIS
   SPTP {A1 5.817, A2 -71.019, A3 88.079, A4 117.546, A5 -39.142, A6 0.000, E1 2440.34, E2 0, E3 0, E4 0, E5 0, E6 0} C_DIS
   SPTP {A1 5.589, A2 -71.520, A3 89.787, A4 114.043, A5 -36.752, A6 0.000, E1 2446.33, E2 0, E3 0, E4 0, E5 0, E6 0} C_DIS
   SPTP {A1 5.374, A2 -71.925, A3 91.409, A4 109.922, A5 -34.586, A6 0.000, E1 2452.91, E2 0, E3 0, E4 0, E5 0, E6 0} C_DIS
   SPTP {A1 5.170, A2 -72.234, A3 92.942, A4 105.145, A5 -32.691, A6 0.000, E1 2460.11, E2 0, E3 0, E4 0, E5 0, E6 0} C_DIS
   SPTP {A1 4.980, A2 -72.443, A3 94.377, A4 99.718, A5 -31.134, A6 0.000, E1 2467.93, E2 0, E3 0, E4 0, E5 0, E6 0} C_DIS
   SPTP {A1 4.807, A2 -72.532, A3 95.802, A4 93.121, A5 -30.002, A6 0.000, E1 2476.88, E2 0, E3 0, E4 0, E5 0, E6 0} C_DIS
   SPTP {A1 4.642, A2 -72.476, A3 97.215, A4 85.309, A5 -29.457, A6 0.000, E1 2486.98, E2 0, E3 0, E4 0, E5 0, E6 0} C_DIS
   SPTP {A1 4.484, A2 -72.289, A3 98.482, A4 77.363, A5 -29.547, A6 0.000, E1 2497.19, E2 0, E3 0, E4 0, E5 0, E6 0} C_DIS
   SPTP {A1 4.334, A2 -71.971, A3 99.599, A4 69.657, A5 -30.263, A6 0.000, E1 2507.14, E2 0, E3 0, E4 0, E5 0, E6 0} C_DIS
   SPTP {A1 4.194, A2 -71.527, A3 100.561, A4 62.514, A5 -31.557, A6 0.000, E1 2516.53, E2 0, E3 0, E4 0, E5 0, E6 0} C_DIS
   SPTP {A1 4.067, A2 -70.955, A3 101.362, A4 56.149, A5 -33.356, A6 0.000, E1 2525.14, E2 0, E3 0, E4 0, E5 0, E6 0} C_DIS
   SPTP {A1 3.955, A2 -70.264, A3 101.997, A4 50.638, A5 -35.562, A6 0.000, E1 2532.9, E2 0, E3 0, E4 0, E5 0, E6 0} C_DIS
   SPTP {A1 3.856, A2 -69.460, A3 102.469, A4 45.950, A5 -38.081, A6 0.000, E1 2539.85, E2 0, E3 0, E4 0, E5 0, E6 0} C_DIS
   SPTP {A1 3.775, A2 -68.549, A3 102.772, A4 42.030, A5 -40.833, A6 0.000, E1 2546.05, E2 0, E3 0, E4 0, E5 0, E6 0} C_DIS
   SPTP {A1 3.713, A2 -67.549, A3 102.906, A4 38.822, A5 -43.722, A6 0.000, E1 2551.56, E2 0, E3 0, E4 0, E5 0, E6 0} C_DIS
   SPTP {A1 3.662, A2 -66.819, A3 102.960, A4 36.789, A5 -45.836, A6 0.000, E1 2555.6, E2 0, E3 0, E4 0, E5 0, E6 0} C_DIS
   SPTP {A1 3.633, A2 -66.042, A3 102.920, A4 35.077, A5 -48.002, A6 0.000, E1 2559.35, E2 0, E3 0, E4 0, E5 0, E6 0} C_DIS
   SPTP {A1 3.622, A2 -65.220, A3 102.788, A4 33.648, A5 -50.198, A6 0.000, E1 2562.86, E2 0, E3 0, E4 0, E5 0, E6 0} C_DIS
   SPTP {A1 3.630, A2 -64.360, A3 102.564, A4 32.473, A5 -52.409, A6 0.000, E1 2566.14, E2 0, E3 0, E4 0, E5 0, E6 0} C_DIS
   SPTP {A1 3.658, A2 -63.462, A3 102.249, A4 31.531, A5 -54.622, A6 0.000, E1 2569.23, E2 0, E3 0, E4 0, E5 0, E6 0} C_DIS
   SPTP {A1 3.706, A2 -62.532, A3 101.843, A4 30.800, A5 -56.823, A6 0.000, E1 2572.14, E2 0, E3 0, E4 0, E5 0, E6 0} C_DIS
   SPTP {A1 3.794, A2 -61.815, A3 101.472, A4 30.495, A5 -58.493, A6 0.000, E1 2574.64, E2 0, E3 0, E4 0, E5 0, E6 0} C_DIS
   SPTP {A1 3.921, A2 -61.308, A3 101.166, A4 30.534, A5 -59.679, A6 0.000, E1 2576.8, E2 0, E3 0, E4 0, E5 0, E6 0} C_DIS
   SPTP {A1 4.065, A2 -60.792, A3 100.819, A4 30.680, A5 -60.853, A6 0.000, E1 2578.88, E2 0, E3 0, E4 0, E5 0, E6 0} C_DIS
   SPTP {A1 4.224, A2 -60.267, A3 100.433, A4 30.924, A5 -62.012, A6 0.000, E1 2580.88, E2 0, E3 0, E4 0, E5 0, E6 0} C_DIS
   SPTP {A1 4.394, A2 -59.736, A3 100.013, A4 31.241, A5 -63.151, A6 0.000, E1 2582.84, E2 0, E3 0, E4 0, E5 0, E6 0} C_DIS
   SPTP {A1 4.574, A2 -59.199, A3 99.556, A4 31.634, A5 -64.269, A6 0.000, E1 2584.75, E2 0, E3 0, E4 0, E5 0, E6 0} C_DIS
   SPTP {A1 4.765, A2 -58.657, A3 99.063, A4 32.098, A5 -65.365, A6 0.000, E1 2586.6, E2 0, E3 0, E4 0, E5 0, E6 0} C_DIS
   SPTP {A1 4.962, A2 -58.111, A3 98.536, A4 32.621, A5 -66.437, A6 0.000, E1 2588.41, E2 0, E3 0, E4 0, E5 0, E6 0} C_DIS
   SPTP {A1 5.215, A2 -57.833, A3 98.149, A4 33.478, A5 -66.969, A6 0.000, E1 2589.95, E2 0, E3 0, E4 0, E5 0, E6 0} C_DIS
   SPTP {A1 5.493, A2 -57.662, A3 97.804, A4 34.497, A5 -67.283, A6 0.000, E1 2591.36, E2 0, E3 0, E4 0, E5 0, E6 0} C_DIS
   SPTP {A1 5.774, A2 -57.489, A3 97.437, A4 35.556, A5 -67.585, A6 0.000, E1 2592.73, E2 0, E3 0, E4 0, E5 0, E6 0} C_DIS
   SPTP {A1 6.058, A2 -57.314, A3 97.046, A4 36.650, A5 -67.874, A6 0.000, E1 2594.06, E2 0, E3 0, E4 0, E5 0, E6 0} C_DIS
   SPTP {A1 6.343, A2 -57.135, A3 96.633, A4 37.775, A5 -68.154, A6 0.000, E1 2595.37, E2 0, E3 0, E4 0, E5 0, E6 0} C_DIS
   SPTP {A1 6.628, A2 -56.954, A3 96.196, A4 38.929, A5 -68.424, A6 0.000, E1 2596.64, E2 0, E3 0, E4 0, E5 0, E6 0} C_DIS
   SPTP {A1 6.912, A2 -56.770, A3 95.738, A4 40.105, A5 -68.683, A6 0.000, E1 2597.9, E2 0, E3 0, E4 0, E5 0, E6 0} C_DIS
   SPTP {A1 7.193, A2 -56.584, A3 95.259, A4 41.299, A5 -68.932, A6 0.000, E1 2599.12, E2 0, E3 0, E4 0, E5 0, E6 0} C_DIS
   SPTP {A1 7.471, A2 -56.397, A3 94.760, A4 42.507, A5 -69.171, A6 0.000, E1 2600.34, E2 0, E3 0, E4 0, E5 0, E6 0} C_DIS
   SPTP {A1 7.744, A2 -56.208, A3 94.243, A4 43.726, A5 -69.399, A6 0.000, E1 2601.53, E2 0, E3 0, E4 0, E5 0, E6 0} C_DIS
   SPTP {A1 8.011, A2 -56.020, A3 93.711, A4 44.949, A5 -69.614, A6 0.000, E1 2602.71, E2 0, E3 0, E4 0, E5 0, E6 0} C_DIS
   SPTP {A1 8.272, A2 -55.832, A3 93.164, A4 46.176, A5 -69.818, A6 0.000, E1 2603.89, E2 0, E3 0, E4 0, E5 0, E6 0} C_DIS
   SPTP {A1 8.538, A2 -55.764, A3 92.689, A4 47.523, A5 -69.811, A6 0.000, E1 2604.86, E2 0, E3 0, E4 0, E5 0, E6 0} C_DIS
   SPTP {A1 8.798, A2 -55.697, A3 92.200, A4 48.879, A5 -69.794, A6 0.000, E1 2605.82, E2 0, E3 0, E4 0, E5 0, E6 0} C_DIS
   SPTP {A1 9.049, A2 -55.629, A3 91.697, A4 50.235, A5 -69.771, A6 0.000, E1 2606.76, E2 0, E3 0, E4 0, E5 0, E6 0} C_DIS
   SPTP {A1 9.292, A2 -55.560, A3 91.181, A4 51.590, A5 -69.745, A6 0.000, E1 2607.69, E2 0, E3 0, E4 0, E5 0, E6 0} C_DIS
   SPTP {A1 9.526, A2 -55.491, A3 90.655, A4 52.941, A5 -69.712, A6 0.000, E1 2608.62, E2 0, E3 0, E4 0, E5 0, E6 0} C_DIS
   SPTP {A1 9.751, A2 -55.422, A3 90.119, A4 54.288, A5 -69.675, A6 0.000, E1 2609.54, E2 0, E3 0, E4 0, E5 0, E6 0} C_DIS
   SPTP {A1 9.966, A2 -55.356, A3 89.576, A4 55.625, A5 -69.631, A6 0.000, E1 2610.45, E2 0, E3 0, E4 0, E5 0, E6 0} C_DIS
   SPTP {A1 10.170, A2 -55.292, A3 89.029, A4 56.952, A5 -69.580, A6 0.000, E1 2611.37, E2 0, E3 0, E4 0, E5 0, E6 0} C_DIS
   SPTP {A1 10.364, A2 -55.231, A3 88.479, A4 58.267, A5 -69.521, A6 0.000, E1 2612.29, E2 0, E3 0, E4 0, E5 0, E6 0} C_DIS
   SPTP {A1 10.548, A2 -55.175, A3 87.929, A4 59.569, A5 -69.452, A6 0.000, E1 2613.2, E2 0, E3 0, E4 0, E5 0, E6 0} C_DIS
   SPTP {A1 10.710, A2 -55.126, A3 87.407, A4 60.802, A5 -69.393, A6 0.000, E1 2614.11, E2 0, E3 0, E4 0, E5 0, E6 0} C_DIS
   SPTP {A1 10.859, A2 -55.084, A3 86.896, A4 62.006, A5 -69.326, A6 0.000, E1 2615.01, E2 0, E3 0, E4 0, E5 0, E6 0} C_DIS
   SPTP {A1 10.971, A2 -55.052, A3 86.461, A4 63.043, A5 -69.299, A6 0.000, E1 2615.86, E2 0, E3 0, E4 0, E5 0, E6 0} C_DIS
   SPTP {A1 11.074, A2 -55.028, A3 86.038, A4 64.059, A5 -69.260, A6 0.000, E1 2616.73, E2 0, E3 0, E4 0, E5 0, E6 0} C_DIS
   SPTP {A1 11.169, A2 -55.014, A3 85.626, A4 65.057, A5 -69.207, A6 0.000, E1 2617.61, E2 0, E3 0, E4 0, E5 0, E6 0} C_DIS
   SPTP {A1 11.256, A2 -55.011, A3 85.230, A4 66.036, A5 -69.138, A6 0.000, E1 2618.5, E2 0, E3 0, E4 0, E5 0, E6 0} C_DIS
   SPTP {A1 11.334, A2 -55.019, A3 84.849, A4 66.995, A5 -69.051, A6 0.000, E1 2619.41, E2 0, E3 0, E4 0, E5 0, E6 0} C_DIS
   SPTP {A1 11.404, A2 -55.040, A3 84.485, A4 67.935, A5 -68.947, A6 0.000, E1 2620.33, E2 0, E3 0, E4 0, E5 0, E6 0} C_DIS
   SPTP {A1 11.466, A2 -55.074, A3 84.141, A4 68.853, A5 -68.822, A6 0.000, E1 2621.26, E2 0, E3 0, E4 0, E5 0, E6 0} C_DIS
   SPTP {A1 11.519, A2 -55.123, A3 83.818, A4 69.751, A5 -68.675, A6 0.000, E1 2622.21, E2 0, E3 0, E4 0, E5 0, E6 0} C_DIS
   SPTP {A1 11.565, A2 -55.186, A3 83.517, A4 70.628, A5 -68.506, A6 0.000, E1 2623.18, E2 0, E3 0, E4 0, E5 0, E6 0} C_DIS
   SPTP {A1 11.602, A2 -55.264, A3 83.239, A4 71.484, A5 -68.315, A6 0.000, E1 2624.16, E2 0, E3 0, E4 0, E5 0, E6 0} C_DIS
   SPTP {A1 11.631, A2 -55.359, A3 82.987, A4 72.319, A5 -68.100, A6 0.000, E1 2625.16, E2 0, E3 0, E4 0, E5 0, E6 0} C_DIS
   SPTP {A1 11.653, A2 -55.469, A3 82.761, A4 73.133, A5 -67.860, A6 0.000, E1 2626.17, E2 0, E3 0, E4 0, E5 0, E6 0} C_DIS
   SPTP {A1 11.666, A2 -55.596, A3 82.561, A4 73.926, A5 -67.594, A6 0.000, E1 2627.2, E2 0, E3 0, E4 0, E5 0, E6 0} C_DIS
   SPTP {A1 11.672, A2 -55.740, A3 82.388, A4 74.698, A5 -67.301, A6 0.000, E1 2628.25, E2 0, E3 0, E4 0, E5 0, E6 0} C_DIS
   SPTP {A1 11.669, A2 -55.901, A3 82.244, A4 75.448, A5 -66.980, A6 0.000, E1 2629.31, E2 0, E3 0, E4 0, E5 0, E6 0} C_DIS
   SPTP {A1 11.659, A2 -56.080, A3 82.131, A4 76.176, A5 -66.629, A6 0.000, E1 2630.39, E2 0, E3 0, E4 0, E5 0, E6 0} C_DIS
   SPTP {A1 11.641, A2 -56.277, A3 82.045, A4 76.885, A5 -66.251, A6 0.000, E1 2631.49, E2 0, E3 0, E4 0, E5 0, E6 0} C_DIS
   SPTP {A1 11.607, A2 -56.543, A3 82.049, A4 77.607, A5 -65.809, A6 0.000, E1 2632.29, E2 0, E3 0, E4 0, E5 0, E6 0} C_DIS
   SPTP {A1 11.566, A2 -56.822, A3 82.075, A4 78.317, A5 -65.346, A6 0.000, E1 2633.08, E2 0, E3 0, E4 0, E5 0, E6 0} C_DIS
   SPTP {A1 11.517, A2 -57.113, A3 82.120, A4 79.015, A5 -64.860, A6 0.000, E1 2633.88, E2 0, E3 0, E4 0, E5 0, E6 0} C_DIS
   SPTP {A1 11.462, A2 -57.417, A3 82.187, A4 79.698, A5 -64.349, A6 0.000, E1 2634.69, E2 0, E3 0, E4 0, E5 0, E6 0} C_DIS
   SPTP {A1 11.398, A2 -57.733, A3 82.275, A4 80.368, A5 -63.813, A6 0.000, E1 2635.51, E2 0, E3 0, E4 0, E5 0, E6 0} C_DIS
   SPTP {A1 11.328, A2 -58.062, A3 82.385, A4 81.023, A5 -63.251, A6 0.000, E1 2636.33, E2 0, E3 0, E4 0, E5 0, E6 0} C_DIS
   SPTP {A1 11.249, A2 -58.404, A3 82.517, A4 81.663, A5 -62.662, A6 0.000, E1 2637.15, E2 0, E3 0, E4 0, E5 0, E6 0} C_DIS
   SPTP {A1 11.163, A2 -58.759, A3 82.670, A4 82.289, A5 -62.044, A6 0.000, E1 2637.99, E2 0, E3 0, E4 0, E5 0, E6 0} C_DIS
   SPTP {A1 11.068, A2 -59.125, A3 82.844, A4 82.900, A5 -61.399, A6 0.000, E1 2638.82, E2 0, E3 0, E4 0, E5 0, E6 0} C_DIS
   SPTP {A1 10.965, A2 -59.503, A3 83.039, A4 83.498, A5 -60.727, A6 0.000, E1 2639.66, E2 0, E3 0, E4 0, E5 0, E6 0} C_DIS
   SPTP {A1 10.854, A2 -59.892, A3 83.254, A4 84.082, A5 -60.024, A6 0.000, E1 2640.51, E2 0, E3 0, E4 0, E5 0, E6 0} C_DIS
   SPTP {A1 10.735, A2 -60.299, A3 83.479, A4 84.701, A5 -59.280, A6 0.000, E1 2641.3, E2 0, E3 0, E4 0, E5 0, E6 0} C_DIS
   SPTP {A1 10.614, A2 -60.771, A3 83.616, A4 85.796, A5 -58.393, A6 0.000, E1 2641.54, E2 0, E3 0, E4 0, E5 0, E6 0} C_DIS
   SPTP {A1 10.482, A2 -61.246, A3 83.757, A4 86.904, A5 -57.493, A6 0.000, E1 2641.76, E2 0, E3 0, E4 0, E5 0, E6 0} C_DIS
   SPTP {A1 10.338, A2 -61.723, A3 83.905, A4 88.025, A5 -56.578, A6 0.000, E1 2641.95, E2 0, E3 0, E4 0, E5 0, E6 0} C_DIS
   SPTP {A1 10.183, A2 -62.202, A3 84.057, A4 89.159, A5 -55.649, A6 0.000, E1 2642.11, E2 0, E3 0, E4 0, E5 0, E6 0} C_DIS
   SPTP {A1 10.016, A2 -62.680, A3 84.214, A4 90.310, A5 -54.710, A6 0.000, E1 2642.25, E2 0, E3 0, E4 0, E5 0, E6 0} C_DIS
   SPTP {A1 9.837, A2 -63.158, A3 84.373, A4 91.480, A5 -53.759, A6 0.000, E1 2642.35, E2 0, E3 0, E4 0, E5 0, E6 0} C_DIS
   SPTP {A1 9.647, A2 -63.636, A3 84.536, A4 92.671, A5 -52.797, A6 0.000, E1 2642.42, E2 0, E3 0, E4 0, E5 0, E6 0} C_DIS
   SPTP {A1 9.445, A2 -64.113, A3 84.702, A4 93.885, A5 -51.825, A6 0.000, E1 2642.46, E2 0, E3 0, E4 0, E5 0, E6 0} C_DIS
   SPTP {A1 9.230, A2 -64.589, A3 84.871, A4 95.125, A5 -50.842, A6 0.000, E1 2642.46, E2 0, E3 0, E4 0, E5 0, E6 0} C_DIS
   SPTP {A1 9.004, A2 -65.062, A3 85.042, A4 96.394, A5 -49.851, A6 0.000, E1 2642.41, E2 0, E3 0, E4 0, E5 0, E6 0} C_DIS
   SPTP {A1 8.765, A2 -65.533, A3 85.215, A4 97.694, A5 -48.851, A6 0.000, E1 2642.32, E2 0, E3 0, E4 0, E5 0, E6 0} C_DIS
   SPTP {A1 8.514, A2 -66.001, A3 85.389, A4 99.029, A5 -47.844, A6 0.000, E1 2642.19, E2 0, E3 0, E4 0, E5 0, E6 0} C_DIS
   SPTP {A1 8.251, A2 -66.465, A3 85.562, A4 100.403, A5 -46.833, A6 0.000, E1 2642.01, E2 0, E3 0, E4 0, E5 0, E6 0} C_DIS
   SPTP {A1 7.976, A2 -66.923, A3 85.736, A4 101.820, A5 -45.821, A6 0.000, E1 2641.77, E2 0, E3 0, E4 0, E5 0, E6 0} C_DIS
   SPTP {A1 7.686, A2 -67.378, A3 85.872, A4 103.428, A5 -44.787, A6 0.000, E1 2641.4, E2 0, E3 0, E4 0, E5 0, E6 0} C_DIS
   SPTP {A1 7.372, A2 -67.834, A3 85.932, A4 105.427, A5 -43.704, A6 0.000, E1 2640.79, E2 0, E3 0, E4 0, E5 0, E6 0} C_DIS
   SPTP {A1 7.043, A2 -68.278, A3 85.988, A4 107.504, A5 -42.641, A6 0.000, E1 2640.1, E2 0, E3 0, E4 0, E5 0, E6 0} C_DIS
   SPTP {A1 6.699, A2 -68.712, A3 86.041, A4 109.662, A5 -41.598, A6 0.000, E1 2639.31, E2 0, E3 0, E4 0, E5 0, E6 0} C_DIS
   SPTP {A1 6.341, A2 -69.134, A3 86.091, A4 111.908, A5 -40.581, A6 0.000, E1 2638.43, E2 0, E3 0, E4 0, E5 0, E6 0} C_DIS
   SPTP {A1 5.969, A2 -69.544, A3 86.137, A4 114.244, A5 -39.590, A6 0.000, E1 2637.45, E2 0, E3 0, E4 0, E5 0, E6 0} C_DIS
   SPTP {A1 5.585, A2 -69.939, A3 86.177, A4 116.676, A5 -38.638, A6 0.000, E1 2636.38, E2 0, E3 0, E4 0, E5 0, E6 0} C_DIS
   SPTP {A1 5.190, A2 -70.320, A3 86.212, A4 119.204, A5 -37.730, A6 0.000, E1 2635.2, E2 0, E3 0, E4 0, E5 0, E6 0} C_DIS
   SPTP {A1 4.785, A2 -70.685, A3 86.239, A4 121.828, A5 -36.874, A6 0.000, E1 2633.93, E2 0, E3 0, E4 0, E5 0, E6 0} C_DIS
   SPTP {A1 4.372, A2 -71.033, A3 86.260, A4 124.546, A5 -36.074, A6 0.000, E1 2632.57, E2 0, E3 0, E4 0, E5 0, E6 0} C_DIS
   SPTP {A1 3.953, A2 -71.364, A3 86.273, A4 127.352, A5 -35.338, A6 0.000, E1 2631.12, E2 0, E3 0, E4 0, E5 0, E6 0} C_DIS
   SPTP {A1 3.526, A2 -71.679, A3 86.282, A4 130.243, A5 -34.665, A6 0.000, E1 2629.6, E2 0, E3 0, E4 0, E5 0, E6 0} C_DIS
   SPTP {A1 3.094, A2 -71.979, A3 86.286, A4 133.208, A5 -34.060, A6 0.000, E1 2628, E2 0, E3 0, E4 0, E5 0, E6 0} C_DIS
   SPTP {A1 2.661, A2 -72.260, A3 86.282, A4 136.229, A5 -33.536, A6 0.000, E1 2626.37, E2 0, E3 0, E4 0, E5 0, E6 0} C_DIS
   SPTP {A1 2.226, A2 -72.601, A3 86.561, A4 138.699, A5 -32.633, A6 0.000, E1 2625.43, E2 0, E3 0, E4 0, E5 0, E6 0} C_DIS
   SPTP {A1 1.791, A2 -72.973, A3 87.006, A4 140.904, A5 -31.500, A6 0.000, E1 2624.84, E2 0, E3 0, E4 0, E5 0, E6 0} C_DIS
   SPTP {A1 1.358, A2 -73.334, A3 87.458, A4 143.190, A5 -30.391, A6 0.000, E1 2624.17, E2 0, E3 0, E4 0, E5 0, E6 0} C_DIS
   SPTP {A1 0.931, A2 -73.683, A3 87.916, A4 145.555, A5 -29.308, A6 0.000, E1 2623.43, E2 0, E3 0, E4 0, E5 0, E6 0} C_DIS
   SPTP {A1 0.513, A2 -74.020, A3 88.381, A4 147.978, A5 -28.262, A6 0.000, E1 2622.65, E2 0, E3 0, E4 0, E5 0, E6 0} C_DIS
   SPTP {A1 0.110, A2 -74.345, A3 88.851, A4 150.446, A5 -27.254, A6 0.000, E1 2621.84, E2 0, E3 0, E4 0, E5 0, E6 0} C_DIS
   SPTP {A1 -0.274, A2 -74.658, A3 89.326, A4 152.928, A5 -26.291, A6 0.000, E1 2621.04, E2 0, E3 0, E4 0, E5 0, E6 0} C_DIS
   SPTP {A1 -0.631, A2 -75.026, A3 90.093, A4 154.785, A5 -24.833, A6 0.000, E1 2620.88, E2 0, E3 0, E4 0, E5 0, E6 0} C_DIS
   SPTP {A1 -0.956, A2 -75.465, A3 91.285, A4 155.622, A5 -22.569, A6 0.000, E1 2621.76, E2 0, E3 0, E4 0, E5 0, E6 0} C_DIS
   SPTP {A1 -1.249, A2 -75.868, A3 92.459, A4 156.320, A5 -20.313, A6 0.000, E1 2622.78, E2 0, E3 0, E4 0, E5 0, E6 0} C_DIS
   SPTP {A1 -1.507, A2 -76.236, A3 93.614, A4 156.800, A5 -18.063, A6 0.000, E1 2624.04, E2 0, E3 0, E4 0, E5 0, E6 0} C_DIS
   SPTP {A1 -1.722, A2 -76.568, A3 94.750, A4 156.899, A5 -15.828, A6 0.000, E1 2625.71, E2 0, E3 0, E4 0, E5 0, E6 0} C_DIS
   SPTP {A1 -1.884, A2 -76.886, A3 96.157, A4 154.944, A5 -12.953, A6 0.000, E1 2629.44, E2 0, E3 0, E4 0, E5 0, E6 0} C_DIS
   SPTP {A1 -2.001, A2 -77.146, A3 97.978, A4 147.046, A5 -9.085, A6 0.000, E1 2639.07, E2 0, E3 0, E4 0, E5 0, E6 0} C_DIS
   SPTP {A1 -2.062, A2 -77.278, A3 99.678, A4 127.215, A5 -5.760, A6 0.000, E1 2660.65, E2 0, E3 0, E4 0, E5 0, E6 0} C_DIS
   SPTP {A1 -2.075, A2 -77.281, A3 101.257, A4 81.174, A5 -4.447, A6 0.000, E1 2708.44, E2 0, E3 0, E4 0, E5 0, E6 0} C_DIS
   SPTP {A1 -2.028, A2 -77.152, A3 102.705, A4 42.164, A5 -6.560, A6 0.000, E1 2749.23, E2 0, E3 0, E4 0, E5 0, E6 0} C_DIS
   SPTP {A1 -1.948, A2 -76.629, A3 104.497, A4 22.366, A5 -12.011, A6 0.000, E1 2770.82, E2 0, E3 0, E4 0, E5 0, E6 0} C_DIS
   SPTP {A1 -1.827, A2 -75.785, A3 106.010, A4 15.665, A5 -18.224, A6 0.000, E1 2779.31, E2 0, E3 0, E4 0, E5 0, E6 0} C_DIS
   SPTP {A1 -1.672, A2 -74.651, A3 107.169, A4 12.822, A5 -24.538, A6 0.000, E1 2783.94, E2 0, E3 0, E4 0, E5 0, E6 0} C_DIS
   SPTP {A1 -1.495, A2 -72.956, A3 108.024, A4 11.022, A5 -31.851, A6 0.000, E1 2787.67, E2 0, E3 0, E4 0, E5 0, E6 0} C_DIS
   SPTP {A1 -1.302, A2 -70.555, A3 108.342, A4 9.871, A5 -40.123, A6 0.000, E1 2790.93, E2 0, E3 0, E4 0, E5 0, E6 0} C_DIS
   SPTP {A1 -1.103, A2 -67.776, A3 107.970, A4 9.354, A5 -48.119, A6 0.000, E1 2793.57, E2 0, E3 0, E4 0, E5 0, E6 0} C_DIS
   SPTP {A1 -0.911, A2 -64.695, A3 106.911, A4 9.169, A5 -55.747, A6 0.000, E1 2795.9, E2 0, E3 0, E4 0, E5 0, E6 0} C_DIS
   SPTP {A1 -0.645, A2 -61.673, A3 105.343, A4 9.432, A5 -62.357, A6 0.000, E1 2798.16, E2 0, E3 0, E4 0, E5 0, E6 0} C_DIS
   SPTP {A1 -0.223, A2 -59.027, A3 103.570, A4 10.288, A5 -67.597, A6 0.000, E1 2800.48, E2 0, E3 0, E4 0, E5 0, E6 0} C_DIS
   SPTP {A1 0.214, A2 -56.332, A3 101.407, A4 11.285, A5 -72.475, A6 0.000, E1 2802.77, E2 0, E3 0, E4 0, E5 0, E6 0} C_DIS
   SPTP {A1 0.666, A2 -53.611, A3 98.869, A4 12.435, A5 -76.980, A6 0.000, E1 2805.02, E2 0, E3 0, E4 0, E5 0, E6 0} C_DIS
   SPTP {A1 1.126, A2 -50.886, A3 95.977, A4 13.703, A5 -81.106, A6 0.000, E1 2807.25, E2 0, E3 0, E4 0, E5 0, E6 0} C_DIS
   SPTP {A1 1.591, A2 -48.169, A3 92.743, A4 15.092, A5 -84.852, A6 0.000, E1 2809.45, E2 0, E3 0, E4 0, E5 0, E6 0} C_DIS
   SPTP {A1 2.059, A2 -45.461, A3 89.175, A4 16.603, A5 -88.228, A6 0.000, E1 2811.62, E2 0, E3 0, E4 0, E5 0, E6 0} C_DIS
   SPTP {A1 2.530, A2 -42.757, A3 85.270, A4 18.236, A5 -91.243, A6 0.000, E1 2813.73, E2 0, E3 0, E4 0, E5 0, E6 0} C_DIS
   SPTP {A1 2.999, A2 -40.044, A3 81.019, A4 19.978, A5 -93.903, A6 0.000, E1 2815.77, E2 0, E3 0, E4 0, E5 0, E6 0} C_DIS
   SPTP {A1 3.462, A2 -37.300, A3 76.396, A4 21.817, A5 -96.219, A6 0.000, E1 2817.72, E2 0, E3 0, E4 0, E5 0, E6 0} C_DIS
   SPTP {A1 3.931, A2 -34.862, A3 71.973, A4 23.763, A5 -97.937, A6 0.000, E1 2819.47, E2 0, E3 0, E4 0, E5 0, E6 0} C_DIS
   SPTP {A1 4.498, A2 -34.748, A3 71.251, A4 25.954, A5 -97.858, A6 0.000, E1 2820.72, E2 0, E3 0, E4 0, E5 0, E6 0} C_DIS
   SPTP {A1 5.057, A2 -34.614, A3 70.439, A4 28.209, A5 -97.745, A6 0.000, E1 2821.81, E2 0, E3 0, E4 0, E5 0, E6 0} C_DIS
   SPTP {A1 5.605, A2 -34.455, A3 69.533, A4 30.513, A5 -97.606, A6 0.000, E1 2822.75, E2 0, E3 0, E4 0, E5 0, E6 0} C_DIS
   SPTP {A1 6.116, A2 -34.675, A3 69.259, A4 32.740, A5 -97.211, A6 0.000, E1 2823.42, E2 0, E3 0, E4 0, E5 0, E6 0} C_DIS
   SPTP {A1 6.593, A2 -35.306, A3 69.675, A4 34.884, A5 -96.536, A6 0.000, E1 2823.77, E2 0, E3 0, E4 0, E5 0, E6 0} C_DIS
   SPTP {A1 7.020, A2 -35.841, A3 69.947, A4 36.871, A5 -95.912, A6 0.000, E1 2823.98, E2 0, E3 0, E4 0, E5 0, E6 0} C_DIS
   SPTP {A1 7.439, A2 -36.344, A3 70.130, A4 38.875, A5 -95.282, A6 0.000, E1 2824.11, E2 0, E3 0, E4 0, E5 0, E6 0} C_DIS
   SPTP {A1 7.440, A2 -36.329, A3 70.111, A4 38.888, A5 -95.294, A6 0.000, E1 2824.09, E2 0, E3 0, E4 0, E5 0, E6 0} C_DIS
   SPTP {A1 7.887, A2 -36.849, A3 70.224, A4 41.093, A5 -94.600, A6 0.000, E1 2824.17, E2 0, E3 0, E4 0, E5 0, E6 0} C_DIS
